(* IEC 61131-3 sources: volt/packages/volt-lsp-iec/test-corpus/pro2193/Device/Plc Logic/Application/09 Misc/Library Manager/L_MC1P_MotionControlBasic (part 3) *)

(* ---- L_MB1P_TPCONVERTTP.pou ---- *)
FUNCTION_BLOCK L_MB1P_TPCONVERTTP
VAR_INPUT
	XENABLE : BOOL;
	XTPRECEIVE : BOOL;
	LRACTTPPOSIN : LREAL;
	LRCYCPOSTPAXIS : LREAL;
	LRCYCPOSTARGETAXIS : LREAL;
	LRCYCLELENGTHTPAXIS : LREAL;
	LRCYCLELENGTHTARGETAXIS : LREAL;
END_VAR
VAR_OUTPUT
	XTPRECEIVED : BOOL;
	LRTPACTPOS : LREAL;
	XERROR : BOOL;
	EERRORID : L_IE1P_Error;
END_VAR
VAR
	LRPOSFIFOX : ARRAY [1..20] OF LREAL := [10(0)];
	LRPOSFIFOREG : ARRAY [1..20] OF LREAL := [10(0)];
	BYCOUNTER : INT := 1;
	LRSTACKDIFFERENCE : LREAL;
	LRTPDELTAINMS : LREAL;
	LRDELTAPCT : LREAL;
	XTPRECEIVEDOLD : BOOL;
	LRTEMP : LREAL;
	IDIRECTION : INT;
	LRACTTPPOSIN_OLD : LREAL;
	XWAIT : BOOL;
	XWAIT_OLD : BOOL;
	LRACTTPPOSIN_INT : LREAL;
	R_TRIG1 : R_TRIG;
END_VAR
END_FUNCTION_BLOCK

METHOD SEARCHINSTACKNEGATIVE
END_METHOD

METHOD SEARCHINSTACKPOSITIVE
END_METHOD

(* ---- L_MB1P_TPTIMESTAMPTOPOS.pou ---- *)
FUNCTION_BLOCK L_MB1P_TPTIMESTAMPTOPOS
VAR_INPUT
	XENABLE : BOOL;
	XTPRECEIVE : BOOL;
	DWTPTIMESTAMP : DWORD;
	LRACTPOSIN : LREAL;
	LRCYCLELENGTH : LREAL;
	DWDELAYACTPOS : DWORD;
END_VAR
VAR_OUTPUT
	XBUSY : BOOL;
	XERROR : BOOL;
	EERRORID : L_IE1P_Error;
	XTPRECEIVED : BOOL;
	LRTPACTPOS : LREAL;
END_VAR
VAR
	XENABLEOLD : BOOL;
	WACTIDX : WORD;
	ALRPOS : ARRAY [0..31] OF LREAL;
	DITIMESTAMPDIFF : DINT;
	DWACTDCTIME : DWORD;
	DWTASKYCLE_NS : DWORD;
	XINIT : BOOL := TRUE;
	LRBASE : LREAL;
	LRDIFF : LREAL;
	LRFACTOR : LREAL;
	LRCAPTURE : LREAL;
	UDIINTERVAL : UDINT;
	LRINTERVAL : LREAL;
	XTPRECEIVEOLD : BOOL;
	C_WMAXELEMENTS : WORD := 31;
END_VAR
END_FUNCTION_BLOCK

METHOD CALCTPPOS : LREAL
END_METHOD

(* ---- L_MC1P_ABORTTRIGGER_INTERNAL.pou ---- *)
FUNCTION_BLOCK L_MC1P_ABORTTRIGGER_INTERNAL EXTENDS L_MC1P_Template_IntFB
VAR_INPUT
	EXECUTE : BOOL;
	PAUSEACTIVETP : BOOL;
END_VAR
VAR_OUTPUT
	DONE : BOOL;
	BUSY : BOOL;
	ERROR : BOOL;
	ERRORID : L_IE1P_Error;
END_VAR
VAR
	PTPREF : POINTER TO L_MC1P_TPData;
	EXECUTEOLD : BOOL := FALSE;
	SNTPNUMBER : SINT;
END_VAR
END_FUNCTION_BLOCK

METHOD MAIN
VAR_IN_OUT
	AXIS : AXIS_REF;
	FBBASE : L_MC1P_Template_ForAxis;
	TRIGGERINPUT : MC_TRIGGER_REF;
END_VAR
END_METHOD

(* ---- L_MC1P_ADDOFFSETCYCLIC.pou ---- *)
FUNCTION_BLOCK L_MC1P_ADDOFFSETCYCLIC
VAR_INPUT
	LRSETPOS : LREAL;
	LRSETOFFSET : LREAL;
	ETRAVERSINGRANGE : L_MC1P_TraversingRange := L_MC1P_TraversingRange.Modulo;
	LRCYCLELENGTH : LREAL;
END_VAR
VAR_OUTPUT
	LRSETPOSOUT : LREAL;
	XERROR : BOOL;
	EERRORID : L_IE1P_Error;
END_VAR
VAR
	LRPOSDIFF : LREAL;
	LRPOS : LREAL;
	LRLENGTH : LREAL;
END_VAR
END_FUNCTION_BLOCK

(* ---- L_MC1P_AVERAGEFILTERSETVALUES.pou ---- *)
FUNCTION_BLOCK L_MC1P_AVERAGEFILTERSETVALUES EXTENDS L_MC1P_SetSetValueManipulator
VAR_INPUT
	WFILTERDEPTH : WORD;
	XMANIPULATETORQUE : BOOL := FALSE;
END_VAR
VAR_OUTPUT
	XINEQOUT : BOOL;
END_VAR
VAR
	WFILTERDEPTHINT : WORD := 20;
	CWFILTERDEPTHMAX : WORD := 1000;
	LRFILTERDEPTH : LREAL;
	LRINVFILTERDEPTH : LREAL;
	WCOUNTER : WORD;
	XERROR_CHECKINPUTDATA : BOOL;
	LRHOMINGOFFSETACT : LREAL;
	LRFILTEREDPOS : LREAL;
	AVERAGEFILTER : L_MC1P_TimeAverage;
	XMANIPULATETORQUEINT : BOOL := FALSE;
END_VAR
END_FUNCTION_BLOCK

METHOD CALCULATE2
VAR_IN_OUT
	AXIS : AXIS_REF;
END_VAR
END_METHOD

METHOD CALLCYCLIC2
VAR_IN_OUT
	AXIS : AXIS_REF;
END_VAR
END_METHOD

METHOD ENABLEINIT2
VAR_IN_OUT
	AXIS : Axis_REf;
END_VAR
END_METHOD

METHOD INITIALIZEFILTER
END_METHOD

METHOD LOADOFFSET2
VAR_INPUT
	OFFSET : LREAL;
END_VAR
VAR_IN_OUT
	AXIS : AXIS_REF;
END_VAR
END_METHOD

METHOD READINPUTS2
VAR_IN_OUT
	AXIS : AXIS_REF;
END_VAR
END_METHOD

(* ---- L_MC1P_AXIS_REF_POOL_2AXES.pou ---- *)
FUNCTION_BLOCK L_MC1P_AXIS_REF_POOL_2AXES
VAR_OUTPUT
	AXESPOOL : L_MC1P_IAXIS_REF_POOL;
END_VAR
VAR_IN_OUT
	AXIS1 : AXIS_REF;
	AXIS2 : AXIS_REF;
END_VAR
VAR
	AAXIS : ARRAY [1..2] OF POINTER TO AXIS_REF;
	WAXISCOUNT : WORD;
	AXISPOOLCOUNT : WORD;
END_VAR
END_FUNCTION_BLOCK

METHOD GETAXISFROMPOOL : POINTER TO AXIS_REF
VAR_INPUT
	WINDEX : WORD;
END_VAR
END_METHOD

(* ---- L_MC1P_AXIS_REF_POOL_3AXES.pou ---- *)
FUNCTION_BLOCK L_MC1P_AXIS_REF_POOL_3AXES
VAR_OUTPUT
	AXESPOOL : L_MC1P_IAXIS_REF_POOL;
END_VAR
VAR_IN_OUT
	AXIS1 : AXIS_REF;
	AXIS2 : AXIS_REF;
	AXIS3 : AXIS_REF;
END_VAR
VAR
	AAXIS : ARRAY [1..3] OF POINTER TO AXIS_REF;
	WAXISCOUNT : WORD;
	AXISPOOLCOUNT : WORD;
END_VAR
END_FUNCTION_BLOCK

METHOD GETAXISFROMPOOL : POINTER TO AXIS_REF
VAR_INPUT
	WINDEX : WORD;
END_VAR
END_METHOD

(* ---- L_MC1P_AXISBASICCONTROL.pou ---- *)
FUNCTION_BLOCK L_MC1P_AXISBASICCONTROL EXTENDS L_MC1P_Template_Licence_150
VAR_INPUT
	XENABLEINTERNALCONTROL : BOOL;
	XREGULATORON : BOOL;
	XRESETERROR : BOOL;
	XENABLEPOSITIVE : BOOL := TRUE;
	XENABLENEGATIVE : BOOL := TRUE;
	XDISABLESWLIMIT : BOOL := FALSE;
	LROVERRIDE : LREAL := 1.0;
	LROVERRIDEACC : LREAL := 1.0;
	LROVERRIDEJERK : LREAL := 1.0;
	XSTOP : BOOL;
	LRSTOPDEC : LREAL := 360000;
	LRSTOPJERK : LREAL := 0;
	XJOGGINGPOS : BOOL;
	XJOGGINGNEG : BOOL;
	LRJOGGINGSETVEL : LREAL := 3600;
	LRJOGGINGSETACC : LREAL := 36000;
	LRJOGGINGSETDEC : LREAL := 36000;
	LRJOGGINGSETJERK : LREAL := 0;
	XCONTINUOUSUPDATE : BOOL;
	XMOVEVELEXECUTE : BOOL;
	XMOVEABSEXECUTE : BOOL;
	XMOVERELEXECUTE : BOOL;
	XHALT : BOOL;
	LRSETPOS_DIST : LREAL;
	LRSETVEL : LREAL := 3600;
	LRSETACC : LREAL := 36000;
	LRSETDEC : LREAL := 36000;
	LRSETJERK : LREAL := 0;
	ESETDIRECTION : MC_DIRECTION := MC_DIRECTION.mcPositiveDirection;
	XHOMEEXECUTE : BOOL;
	LRHOMEPOSITION : LREAL;
	XUSEHOMEEXTPARAMETER : BOOL;
	SCHOMEEXTPARAMETER : L_MC1P_HomeParameter;
	SCHOMEEXTTP : MC_TRIGGER_REF;
	XHOMEABSSWITCH : BOOL;
END_VAR
VAR_OUTPUT
	XINTERNALCONTROLACTIVE : BOOL;
	XERROR : BOOL;
	EERRORID : L_IE1P_Error;
	XFUNBUSY : BOOL;
	XFUNDONE : BOOL;
	XFUNCOMMANDABORTED : BOOL;
	EFUNSTATEACT : L_MC1P_ABC_State;
	ECONTROLMODE : L_MC1P_ControlMode;
	XISHOMED : BOOL;
	XHWLIMITSWITCHNEG : BOOL;
	XHWLIMITSWITCHPOS : BOOL;
	XSWLIMITENABLED : BOOL;
	XSWLIMITSWITCHNEG : BOOL;
	XSWLIMITSWITCHPOS : BOOL;
	EAXISTYPE : L_MC1P_DriveType;
	EAXISSTATE : L_MC1P_AXIS_STATE := L_MC1P_AXIS_STATE.Disabled;
	XAXISREADY : BOOL;
	XAXISENABLED : BOOL;
	XAXISWARNING : BOOL;
	XAXISERROR : BOOL;
	EAXISERRORID : L_IE1P_Error;
	XDRIVEWARNING : BOOL;
	XDRIVEERROR : BOOL;
	DWDRIVEERRORID : DWORD;
	LRACTPOS : LREAL;
	LRACTVEL : LREAL;
	LRSETPOSOUT : LREAL;
	LRSETVELOUT : LREAL;
	LRACTFOLLOWINGERROR : LREAL;
	XCONSTANTVELOCITY : BOOL;
	XACCELERATING : BOOL;
	XDECELERATING : BOOL;
	XDIRECTIONPOSITIVE : BOOL;
	XDIRECTIONNEGATIVE : BOOL;
	XINPOSITION : BOOL;
	XAXISAVAILABLE : BOOL;
	XSTANDSTILLSETVELOCITY : BOOL;
	XSTANDSTILLACTVELOCITY : BOOL;
	XAXISREADYTOSWITCHON : BOOL;
	XAXISREADYFORMOTION : BOOL;
END_VAR
VAR
	XREGULATORON_INT : BOOL;
	XRESETERROR_INT : BOOL;
	XENABLEPOSITIVE_INT : BOOL;
	XENABLENEGATIVE_INT : BOOL;
	XDISABLESWLIMIT_INT : BOOL;
	LROVERRIDE_INT : LREAL := 1.0;
	LROVERRIDEACC_INT : LREAL := 1.0;
	LROVERRIDEJERK_INT : LREAL := 1.0;
	XSTOP_INT : BOOL;
	LRSTOPDEC_INT : LREAL;
	LRSTOPJERK_INT : LREAL;
	XHALT_INT : BOOL;
	XJOGGINGPOS_INT : BOOL;
	XJOGGINGNEG_INT : BOOL;
	LRJOGGINGSETVEL_INT : LREAL;
	LRJOGGINGSETACC_INT : LREAL;
	LRJOGGINGSETDEC_INT : LREAL;
	LRJOGGINGSETJERK_INT : LREAL := 0;
	LRJOGGINGSETJERKDEC_INT : LREAL := 0;
	LRJOGGINGSETJERKDECAPP : LREAL := 0;
	XMOVEVELEXECUTE_INT : BOOL;
	XMOVEABSEXECUTE_INT : BOOL;
	XMOVERELEXECUTE_INT : BOOL;
	XCONTINUOUSUPDATE_INT : BOOL;
	LRSETPOS_DIST_INT : LREAL;
	LRSETVEL_INT : LREAL;
	LRSETACC_INT : LREAL;
	LRSETDEC_INT : LREAL;
	LRSETJERK_INT : LREAL;
	LRSETJERKDEC_INT : LREAL := 0;
	LRSETJERKDECAPP : LREAL := 0;
	ESETDIRECTION_INT : MC_DIRECTION;
	XHOMEEXECUTE_INT : BOOL;
	LRHOMEPOSITION_INT : LREAL;
	XHOMEEXTERNALVALUES_INT : BOOL;
	SCHOMEEXTPARAMETER_INT : L_MC1P_HomeParameter;
	XDISABLEMOVEFUNEXEC : BOOL;
	XINTERNALCONTROLVISU : BOOL;
	XDISABLEMOVEFUN : BOOL;
	XDISABLEHOMEFUN : BOOL;
	XDISABLEPOWERFUN : BOOL;
	XDISABLEPOWERCALL : BOOL;
	XVISUMOVEFUN : BOOL;
	XVISUHOMEFUN : BOOL;
	XVISUPOWFUN : BOOL;
	ABC : REFERENCE TO L_MC1P_AxisBasicControl_Internal;
	DATA : L_MC1P_AxisBasicControlInstanceData;
	FBBASEOLD : POINTER TO L_MC1P_Template_ForAxis;
	_USEQSP : BOOL := FALSE;
	DISABLEHOMEFUN : BOOL;
	DISABLEMOVEFUN : BOOL;
	DISABLEMOVEFUNEXEC : BOOL;
	DISABLEPOWERCALL : BOOL;
	DISABLEPOWERFUN : BOOL;
	LRJOGGINGSETJERKDEC : LREAL;
	LRSETJERKDEC : LREAL;
	USEQSP : BOOL;
END_VAR
END_FUNCTION_BLOCK

(* ---- L_MC1P_AXISBASICCONTROL_INTERNAL.pou ---- *)
FUNCTION_BLOCK L_MC1P_AXISBASICCONTROL_INTERNAL EXTENDS L_MC1P_Template_IntFB
VAR_INPUT
	XDISABLEPOWERCALL : BOOL;
	XREGULATORON : BOOL;
	XRESETERROR : BOOL;
	XENABLEPOSITIVE : BOOL := TRUE;
	XENABLENEGATIVE : BOOL := TRUE;
	XDISABLESWLIMIT : BOOL;
	LROVERRIDE : LREAL := 1.0;
	LROVERRIDEACC : LREAL := 1.0;
	LROVERRIDEJERK : LREAL := 1.0;
	XSTOP : BOOL;
	LRSTOPDEC : LREAL;
	LRSTOPJERK : LREAL;
	XJOGGINGPOS : BOOL;
	XJOGGINGNEG : BOOL;
	LRJOGGINGSETVEL : LREAL := 3600;
	LRJOGGINGSETACC : LREAL := 36000;
	LRJOGGINGSETDEC : LREAL := 36000;
	LRJOGGINGSETJERK : LREAL := 0;
	LRJOGGINGSETJERKDEC : LREAL := 0;
	XCONTINUOUSUPDATE : BOOL;
	XFINISHPOSITIONING : BOOL;
	XQSPAPPLICATION : BOOL;
	XHALT : BOOL;
	XABORT : BOOL;
	XMOVEVELEXECUTE : BOOL;
	XMOVEABSEXECUTE : BOOL;
	XMOVERELEXECUTE : BOOL;
	LRSETPOS_DIST : LREAL;
	LRSETVEL : LREAL := 3600;
	LRSETACC : LREAL := 36000;
	LRSETDEC : LREAL := 36000;
	LRSETJERK : LREAL := 0;
	LRSETJERKDEC : LREAL := 0;
	ESETDIRECTION : MC_DIRECTION := MC_DIRECTION.mcPositiveDirection;
	XHOMEEXECUTE : BOOL;
	LRHOMEPOSITION : LREAL;
	XUSEHOMEEXTPARAMETER : BOOL;
	SCHOMEEXTPARAMETER : L_MC1P_HomeParameter;
	SCHOMEEXTTP : MC_TRIGGER_REF;
	XHOMEABSSWITCH : BOOL;
	XRESETHOMEPOSITION : BOOL;
	WCALLEDINCYCLE : WORD;
	XQSPDRIVEDONE : BOOL;
	XMOVEVELENABLEOFFSETVEL : BOOL;
	LRMOVEVELOFFSETVEL : LREAL;
	XUSEABORTBEHAVIOURFORTM : BOOL;
	LRABORTDEC : LREAL;
	LRABORTJERK : LREAL;
END_VAR
VAR_OUTPUT
	ECONTROLMODE : L_MC1P_ControlMode;
	XISHOMED : BOOL;
	XHWLIMITSWITCHNEG : BOOL;
	XHWLIMITSWITCHPOS : BOOL;
	XSWLIMITENABLED : BOOL;
	XSWLIMITSWITCHNEG : BOOL;
	XSWLIMITSWITCHPOS : BOOL;
	EAXISTYPE : L_MC1P_DriveType;
	EAXISSTATE : L_MC1P_AXIS_STATE := L_MC1P_AXIS_STATE.Disabled;
	XAXISREADY : BOOL;
	XAXISENABLED : BOOL;
	XAXISWARNING : BOOL;
	XAXISERROR : BOOL;
	EAXISERRORID : L_IE1P_Error;
	XDRIVEWARNING : BOOL;
	XDRIVEERROR : BOOL;
	DWDRIVEERRORID : DWORD;
	LRACTPOS : LREAL;
	LRACTVEL : LREAL;
	LRSETPOSOUT : LREAL;
	LRSETVELOUT : LREAL;
	LRACTFOLLOWINGERROR : LREAL;
	XCONSTANTVELOCITY : BOOL;
	XACCELERATING : BOOL;
	XDECELERATING : BOOL;
	XDIRECTIONPOSITIVE : BOOL;
	XDIRECTIONNEGATIVE : BOOL;
	XINPOSITION : BOOL;
	XAXISAVAILABLE : BOOL;
	XSTANDSTILLSETVELOCITY : BOOL;
	XSTANDSTILLACTVELOCITY : BOOL;
	XAXISREADYTOSWITCHON : BOOL;
	XAXISREADYFORMOTION : BOOL;
END_VAR
VAR
	ABCFUNID : WORD;
	FBSTOP : L_MC1P_Stop_Internal;
	FBHALT : L_MC1P_Halt_Internal;
	FBABORT : L_MC1P_Halt_Internal;
	FBHOME : L_MC1P_Home_Internal;
	FBJOG : L_MC1P_ManualJog_Internal;
	FBMOVEABS : L_MC1P_MoveAbsolute_Inernal;
	FBMOVEVEL : L_MC1P_MoveVelocity_Internal;
	FBMOVEREL : L_MC1P_MoveRelative_Internal;
	FBFINISHPOSITIONING : L_MC1P_FinishPositioning_internal;
	PBDUMMY : POINTER TO BOOL;
	XCONTROLLEDBYAXIS : BOOL;
	XCALLEDBYAXIS : BOOL;
	XUPDATESTATE : BOOL;
	XUPDATECONTROL : BOOL;
	XDISABLEMOVEFUNEXEC : BOOL;
	XDISABLEINTERNALCALLOFMOVEFUNCTIONS : BOOL;
	ETMPHOMEMODE : L_MC1P_HomeMode;
	LRTMPOFFSETPOSITION : LREAL;
	AXISCONTROL : BOOL;
	CALLEDBYAXIS : BOOL;
	DISABLEMOVEFUNEXEC : BOOL;
END_VAR
END_FUNCTION_BLOCK

METHOD BASEITFCHANGED
VAR_INPUT
	FBBASEOLD : POINTER TO POINTER TO L_MC1P_Template_ForAxis;
END_VAR
VAR_IN_OUT
	AXIS : AXIS_REF;
	FBBASE : L_MC1P_Template_ForAxis;
	DATA : L_MC1P_AxisBasicControlInstanceData;
END_VAR
END_METHOD

METHOD CALLMOVEFB : BOOL
VAR_IN_OUT
	AXIS : AXIS_REF;
	DATA : L_MC1P_AxisBasicControlInstanceData;
END_VAR
END_METHOD

METHOD EXITSTATE
VAR_IN_OUT
	AXIS : AXIS_REF;
	DATA : L_MC1P_AxisBasicControlInstanceData;
END_VAR
END_METHOD

METHOD MAIN
VAR_IN_OUT
	AXIS : AXIS_REF;
	FBBASE : L_MC1P_Template_ForAxis;
	DATA : L_MC1P_AxisBasicControlInstanceData;
END_VAR
END_METHOD

METHOD RESET
VAR_IN_OUT
	DATA : L_MC1P_AxisBasicControlInstanceData;
END_VAR
END_METHOD

METHOD RESETACTIVEINSTANCE : WORD
END_METHOD

METHOD SETACTIVEINSTANCE : WORD
END_METHOD

METHOD STATEMACHINE
VAR_IN_OUT
	AXIS : AXIS_REF;
	DATA : L_MC1P_AxisBasicControlInstanceData;
END_VAR
END_METHOD

(* ---- L_MC1P_AXISBASICCONTROLV2.pou ---- *)
FUNCTION_BLOCK L_MC1P_AXISBASICCONTROLV2 EXTENDS L_MC1P_Template_Licence_150
VAR_INPUT
	XENABLEINTERNALCONTROL : BOOL;
	XENABLEOPERATION : BOOL;
	XRESETERROR : BOOL;
	XENABLEPOSITIVE : BOOL := TRUE;
	XENABLENEGATIVE : BOOL := TRUE;
	XDISABLESWLIMIT : BOOL := FALSE;
	LROVERRIDE : LREAL := 1.0;
	LROVERRIDEACC : LREAL := 1.0;
	LROVERRIDEJERK : LREAL := 1.0;
	XQSPAPPLICATION : BOOL;
	XHALT : BOOL;
	XABORT : BOOL;
	XJOGPOS : BOOL;
	XJOGNEG : BOOL;
	XCONTINUOUSUPDATE : BOOL;
	XFINISHPOSITIONING : BOOL;
	XMOVEVELEXECUTE : BOOL;
	XMOVEABSEXECUTE : BOOL;
	XMOVERELEXECUTE : BOOL;
	LRPOS_DIST : LREAL := 0;
	LRVEL : LREAL := 3600;
	LRACC : LREAL := 36000;
	LRDEC : LREAL := 36000;
	LRJERK : LREAL := 0;
	EDIRECTION : MC_DIRECTION := MC_DIRECTION.mcPositiveDirection;
	XHOMEEXECUTE : BOOL;
	SCHOMEEXTTP : MC_TRIGGER_REF;
	XHOMEABSSWITCH : BOOL;
	XRESETHOMEPOSITION : BOOL;
END_VAR
VAR_OUTPUT
	XINTERNALCONTROLACTIVE : BOOL;
	XERROR : BOOL;
	EERRORID : L_IE1P_Error;
	XFUNBUSY : BOOL;
	XFUNDONE : BOOL;
	XFUNCOMMANDABORTED : BOOL;
	EFUNSTATEACT : L_MC1P_ABC_State := L_MC1P_ABC_State.Standby;
	ECONTROLMODE : L_MC1P_ControlMode := L_MC1P_ControlMode.PosCtrlDrive;
	XISHOMED : BOOL;
	XHWLIMITSWITCHNEG : BOOL;
	XHWLIMITSWITCHPOS : BOOL;
	XSWLIMITENABLED : BOOL;
	XSWLIMITSWITCHNEG : BOOL;
	XSWLIMITSWITCHPOS : BOOL;
	EAXISTYPE : L_MC1P_DriveType := L_MC1P_DriveType.Virtual;
	EAXISSTATE : L_MC1P_AXIS_STATE := L_MC1P_AXIS_STATE.Disabled;
	XSTOACTIVE : BOOL;
	XREADYFOROPERATION : BOOL;
	XOPERATIONENABLED : BOOL;
	XREADYFORMOTION : BOOL;
	XAXISWARNING : BOOL;
	XAXISERROR : BOOL;
	EAXISERRORID : L_IE1P_Error;
	XDRIVEWARNING : BOOL;
	XDRIVEERROR : BOOL;
	DWDRIVEERRORID : DWORD;
	LRACTPOS : LREAL;
	LRACTVEL : LREAL;
	LRSETPOSOUT : LREAL;
	LRSETVELOUT : LREAL;
	LRACTFOLLOWINGERROR : LREAL;
	XINPOSITION : BOOL;
	XSTANDSTILLSETVELOCITY : BOOL;
	XSTANDSTILLACTVELOCITY : BOOL;
	XCONSTANTVELOCITY : BOOL;
	XACCELERATING : BOOL;
	XDECELERATING : BOOL;
	XDIRECTIONPOSITIVE : BOOL;
	XDIRECTIONNEGATIVE : BOOL;
	XAXISAVAILABLE : BOOL;
END_VAR
VAR
	_ITFOWNER : L_UBUP.L_UBUP_IFBPool;
	_XWHANDLE : __XWORD;
	_XOCCUPIED : BOOL;
	XENABLEOPERATION_INT : BOOL;
	XRESETERROR_INT : BOOL;
	XENABLEPOSITIVE_INT : BOOL;
	XENABLENEGATIVE_INT : BOOL;
	XDISABLESWLIMIT_INT : BOOL;
	LROVERRIDE_INT : LREAL;
	LROVERRIDEACC_INT : LREAL;
	LROVERRIDEJERK_INT : LREAL;
	XQSPAPPLICATION_INT : BOOL;
	XHALT_INT : BOOL;
	XABORT_INT : BOOL;
	XJOGPOS_INT : BOOL;
	XJOGNEG_INT : BOOL;
	XCONTINUOUSUPDATE_INT : BOOL;
	XFINISHPOSITIONING_INT : BOOL;
	XMOVEVELEXECUTE_INT : BOOL;
	XMOVEABSEXECUTE_INT : BOOL;
	XMOVERELEXECUTE_INT : BOOL;
	LRPOS_DIST_INT : LREAL;
	LRVEL_INT : LREAL;
	LRACC_INT : LREAL;
	LRDEC_INT : LREAL;
	LRJERK_INT : LREAL;
	EDIRECTION_INT : MC_DIRECTION;
	XHOMEEXECUTE_INT : BOOL;
	XRESETHOMEPOSITION_INT : BOOL;
	LRSETJERKDEC_INT : LREAL;
	LRJOGGINGSETJERKDEC_INT : LREAL;
	LRSETJERKDECAPP : LREAL;
	LRJOGGINGSETJERKDECAPP : LREAL;
	XDISABLEMOVEFUNEXEC : BOOL;
	XDISABLEPOWERCALL : BOOL;
	XINTERNALCONTROLVISU : BOOL;
	XDISABLEMOVEFUN : BOOL;
	XDISABLEHOMEFUN : BOOL;
	XDISABLEPOWERFUN : BOOL;
	XVISUMOVEFUN : BOOL;
	XVISUHOMEFUN : BOOL;
	XVISUPOWFUN : BOOL;
	LRMOVEVELOFFSETVELAPP : LREAL;
	XMOVEVELENABLEOFFSETVELAPP : BOOL;
	LRABORTDECAPP : LREAL;
	LRABORTJERKAPP : LREAL;
	XUSEABORTBEHAVIOURFORTM : BOOL;
	ABC : REFERENCE TO L_MC1P_AxisBasicControl_Internal;
	DATA : L_MC1P_AxisBasicControlInstanceData;
	FBBASEOLD : POINTER TO L_MC1P_Template_ForAxis;
	_DWOBJID : DWORD;
	CLASSID : DINT;
	DISABLEHOMEFUN : BOOL;
	DISABLEMOVEFUN : BOOL;
	DISABLEMOVEFUNEXEC : BOOL;
	DISABLEPOWERCALL : BOOL;
	DISABLEPOWERFUN : BOOL;
	INSTANCEPTR : POINTER TO BYTE;
	LRABORTDEC : LREAL;
	LRABORTJERK : LREAL;
	LRJOGGINGSETJERKDEC : LREAL;
	LRMOVEVELOFFSETVEL : LREAL;
	LRSETJERKDEC : LREAL;
	OBJECTID : DWORD;
	OCCUPIED : BOOL;
	REMAININGTIMEOFPROFILE : LREAL;
	REMAININGTIMEOFPROFILEAVAILABLE : BOOL;
	XMOVEVELENABLEOFFSETVEL : BOOL;
	XSPECIALABORTBEHAVIOR : BOOL;
END_VAR
END_FUNCTION_BLOCK

METHOD RESETABORT
END_METHOD

METHOD RESETFINISHPOSITIONING
END_METHOD

METHOD RESETHALT
END_METHOD

METHOD RESETHOMEEXECUTE
END_METHOD

METHOD RESETMOVEABSEXECUTE
END_METHOD

METHOD RESETMOVERELEXECUTE
END_METHOD

METHOD RESETMOVEVELEXECUTE
END_METHOD

METHOD FREE : BOOL
END_METHOD

METHOD OCCUPY : BOOL
VAR_INPUT
	ITFOWNER : L_UBUP.L_UBUP_IFBPool;
	XWHANDLE : __XWORD;
END_VAR
END_METHOD

METHOD REQUESTINTERFACE : BOOL
VAR_INPUT
	ID : DINT;
	PITFUNKNOWN : POINTER TO L_UBUP_IUnknown;
END_VAR
END_METHOD

METHOD FB_INIT : BOOL
VAR_INPUT
	BINITRETAINS : BOOL;
	BINCOPYCODE : BOOL;
END_VAR
END_METHOD

(* ---- L_MC1P_AXISCOMMAND.pou ---- *)
FUNCTION_BLOCK L_MC1P_AXISCOMMAND
VAR_INPUT
	COMMANDIN : USINT;
END_VAR
VAR_OUTPUT
	XCOMMANDBUSY : BOOL;
END_VAR
VAR
	XABORT : BOOL;
	COMMAND : REFERENCE TO USINT;
	COMMANDOLD : USINT;
	FB_BASE : L_MC1P_Template_ForAxis;
	C_CMDREADY : USINT := 0;
	C_CMDSTART : USINT := 1;
	C_CMDINPROGRESS : USINT := 2;
	C_CMDCANCELLED : USINT := 3;
	C_CMDNOACCESS : USINT := 4;
	C_CMDNOACCESSDISABLED : USINT := 5;
	C_CMDABORT : USINT := 16;
	C_CMDWORKING20 : USINT := 20;
	C_CMDWORKING40 : USINT := 40;
	C_CMDWORKING60 : USINT := 60;
	C_CMDWORKING80 : USINT := 80;
	C_CMDWRONGBRAKEMODE : USINT := 101;
	C_CMDSTOACTIVE : USINT := 102;
	C_CMDINVALIDPARAMETERSETTINGS : USINT := 103;
	C_CMDSTARTOUTSIDEPOSLIMITS : USINT := 104;
	C_CMDPOSRANGENOTSUFFICIENT : USINT := 105;
	C_CMDHOMEPOSREQUIRED : USINT := 106;
	C_CMDINVALIDPOSITIONLIMITS : USINT := 107;
	C_CMDVIRTUALMODENOTSUPPORTED : USINT := 120;
	BUSY : BOOL;
END_VAR
END_FUNCTION_BLOCK

METHOD ABORTING
END_METHOD

METHOD CALCSTATUS
VAR_IN_OUT
	AXIS : _AXIS_REF_REAL;
END_VAR
END_METHOD

METHOD EXECUTE
END_METHOD

METHOD MAIN
END_METHOD

METHOD READINPUTS
END_METHOD

METHOD RESETCOMMANDERRORSTATE : BOOL
VAR_IN_OUT
	AXIS : _AXIS_REF_REAL;
END_VAR
END_METHOD

METHOD RESETSTATUSPARAMETER
END_METHOD

METHOD SETINCTANCEINFO
VAR_INPUT
	PSINSTANCENAME : POINTER TO STRING;
	ERRORITFID : DWORD;
END_VAR
END_METHOD

METHOD UPDATEAXISPOINTER
VAR_INPUT
	PAXIS : POINTER TO AXIS_REF;
END_VAR
END_METHOD

METHOD UPDATECOMMANDINTERFACE
VAR_IN_OUT
	CMD : USINT;
END_VAR
END_METHOD

METHOD FB_INIT : BOOL
VAR_INPUT
	BINITRETAINS : BOOL;
	BINCOPYCODE : BOOL;
END_VAR
END_METHOD

(* ---- L_MC1P_AXISCOMMAND_BRAKEGRINDIN.pou ---- *)
FUNCTION_BLOCK L_MC1P_AXISCOMMAND_BRAKEGRINDIN EXTENDS L_MC1P_AxisCommand
VAR_INPUT
	PAXIS : POINTER TO _AXIS_REF_REAL;
	EMODE : L_MC1P_GrindInMode := L_MC1P_GrindInMode.CwCcw;
	LRMOTORSPEED : LREAL := 60.0;
	LRRAMPTIME : LREAL := 1.0;
	LRONTIME : LREAL := 0.5;
	LROFFTIME : LREAL := 0.5;
	WCYCLES : WORD := 4;
	USICONTROL : USINT;
END_VAR
VAR
	FB_BRAKEGRINDIN : L_MC1P_BrakeGrindIn_internal;
	STATUS_100 : LREAL;
	LRSTATUS : LREAL;
	C_WSTATESUCCESSFUL : WORD := 10;
	C_WSTATEABORTEDERROR : WORD := 8;
	C_WSTATEABORTEDUSER : WORD := 9;
END_VAR
END_FUNCTION_BLOCK

METHOD ABORTING
END_METHOD

METHOD EXECUTE
END_METHOD

METHOD READINPUTS
END_METHOD

METHOD RESETSTATUSPARAMETER
END_METHOD

METHOD UPDATEAXISPOINTER
VAR_INPUT
	PAXIS : POINTER TO AXIS_REF;
END_VAR
END_METHOD

(* ---- L_MC1P_AXISCOMMAND_BRAKETEST.pou ---- *)
FUNCTION_BLOCK L_MC1P_AXISCOMMAND_BRAKETEST EXTENDS L_MC1P_AxisCommand
VAR_INPUT
	PAXIS : POINTER TO _AXIS_REF_REAL;
END_VAR
VAR
	FB_BRAKETEST : L_MC1P_BrakeTest_internal;
	ACTPOSTHRESHOLD : INT;
	STATUS_100 : LREAL;
	LRSTATUS : LREAL;
	LRTIME : LREAL;
	C_WSTATESUCCESSFUL : WORD := 10;
	C_WSTATEFAILED : WORD := 11;
	C_WSTATEABORTEDERROR : WORD := 8;
	C_WSTATEABORTEDUSER : WORD := 9;
END_VAR
END_FUNCTION_BLOCK

METHOD ABORTING
END_METHOD

METHOD EXECUTE
END_METHOD

METHOD READINPUTS
END_METHOD

METHOD RESETSTATUSPARAMETER
END_METHOD

METHOD UPDATEAXISPOINTER
VAR_INPUT
	PAXIS : POINTER TO AXIS_REF;
END_VAR
END_METHOD

(* ---- L_MC1P_AXISCONNECTIONVIEWER.pou ---- *)
FUNCTION_BLOCK L_MC1P_AXISCONNECTIONVIEWER EXTENDS L_IF1P_FunctionConnectionViewer
END_FUNCTION_BLOCK

METHOD BUILDUPCONNECTIONTABLE : BOOL
END_METHOD

METHOD FINDCONNECTIONSOURCE : POINTER TO BYTE
VAR_INPUT
	PSLAVECONNECTOR : POINTER TO IoConfigConnector;
	UITYPE : UINT;
	UISUBDEVICE : UINT;
END_VAR
END_METHOD

METHOD FINDFUNCTION : L_IF1P_IFunctionConnection
VAR_INPUT
	PFUNCTIONCONNECTOR : POINTER TO IoConfigConnector;
END_VAR
VAR_OUTPUT
	UITYPE : UINT;
END_VAR
END_METHOD

METHOD GETCONNECTEDSLAVE : BOOL
END_METHOD

METHOD INITIALIZE : UDINT
VAR_INPUT
	WMODULETYPE : UINT;
	DWINSTANCE : UDINT;
	PCONNECTOR : POINTER TO IoConfigConnector;
END_VAR
END_METHOD

METHOD IODRVREADPARAMETER : UDINT
VAR_INPUT
	PCONNECTOR : POINTER TO IoConfigConnector;
	PPARAMETER : POINTER TO IoConfigParameter;
	PDATA : POINTER TO BYTE;
	DWBITSIZE : DWORD;
	DWBITOFFSET : DWORD;
END_VAR
END_METHOD

METHOD IODRVUPDATECONFIGURATION : UDINT
VAR_INPUT
	PCONNECTORLIST : POINTER TO IoConfigConnector;
	NCOUNT : DINT;
END_VAR
END_METHOD

METHOD IODRVUPDATEMAPPING : UDINT
VAR_INPUT
	PTASKMAPLIST : POINTER TO IoConfigTaskMap;
	NCOUNT : DINT;
END_VAR
END_METHOD

METHOD IODRVWRITEPARAMETER : UDINT
VAR_INPUT
	PCONNECTOR : POINTER TO IoConfigConnector;
	PPARAMETER : POINTER TO IoConfigParameter;
	PDATA : POINTER TO BYTE;
	DWBITSIZE : DWORD;
	DWBITOFFSET : DWORD;
END_VAR
END_METHOD

METHOD QUERYINTERFACE : POINTER TO POINTER TO BYTE
VAR_INPUT
	IID : DWORD;
	PRESULT : POINTER TO UDINT;
END_VAR
END_METHOD

METHOD STATUSCHANGED : BOOL
END_METHOD

METHOD FB_EXIT : BOOL
VAR_INPUT
	BINCOPYCODE : BOOL;
END_VAR
END_METHOD

METHOD FB_INIT : BOOL
VAR_INPUT
	BINITRETAINS : BOOL;
	BINCOPYCODE : BOOL;
END_VAR
END_METHOD

METHOD EVENTCALLBACK : UDINT
VAR_INPUT
	PEVENTPARAM : POINTER TO EventParam;
END_VAR
END_METHOD

METHOD REGISTEREVENT
END_METHOD

METHOD UNREGISTEREVENT
END_METHOD

(* ---- L_MC1P_AXISEXTENSION_9400HL.pou ---- *)
FUNCTION_BLOCK L_MC1P_AXISEXTENSION_9400HL EXTENDS L_MC1P_AxisExtensionEmpty
VAR
	ECATCOMM : L_MC1P_CommECAT;
	CONFIGDRIVE : L_MC1P_Config_94HL_ETC;
	DRIVESCALING : L_MC1P_DriveScaling_94HL;
	DRIVESPECIFIC : L_MC1P_DriveSpecific_9400HL;
	FBEXTENDEDMAPPINGACCESS : L_MC1P_ExtendedMappingAccess;
	ITFCOMM : L_MC1P_ICommunication;
	ITFCONFIGDRIVE : L_MC1P_IConfigureDrive;
	ITFDRIVESCALING : L_MC1P_IDriveScaling;
	ITFDRIVESPECIFIC : L_MC1P_IDriveSpecificImplBase;
	ITFEXTENDEDMAPPINGACCESS : L_MC1P_IExtendedMappingAccess;
END_VAR
END_FUNCTION_BLOCK

(* ---- L_MC1P_AXISEXTENSION_9400HL_CAN.pou ---- *)
FUNCTION_BLOCK L_MC1P_AXISEXTENSION_9400HL_CAN EXTENDS L_MC1P_AxisExtensionEmpty
VAR
	CANCOMM : L_MC1P_CommCAN;
	CONFIGDRIVE : L_MC1P_Config_94HL_ETC;
	DRIVESCALING : L_MC1P_DriveScaling_94HL;
	DRIVESPECIFIC : L_MC1P_DriveSpecific_9400HL;
	FBEXTENDEDMAPPINGACCESS : L_MC1P_ExtendedMappingAccess;
	ITFCOMM : L_MC1P_ICommunication;
	ITFCONFIGDRIVE : L_MC1P_IConfigureDrive;
	ITFDRIVESCALING : L_MC1P_IDriveScaling;
	ITFDRIVESPECIFIC : L_MC1P_IDriveSpecificImplBase;
	ITFEXTENDEDMAPPINGACCESS : L_MC1P_IExtendedMappingAccess;
END_VAR
END_FUNCTION_BLOCK

(* ---- L_MC1P_AXISEXTENSION_ENCBPB.pou ---- *)
FUNCTION_BLOCK L_MC1P_AXISEXTENSION_ENCBPB EXTENDS L_MC1P_AxisExtensionEmpty
VAR
	DRIVESPECIFIC : L_MC1P_DriveSpecific_Enc_Bpb;
	DRIVESCALING : L_MC1P_DriveScaling;
	ITFDRIVESCALING : L_MC1P_IDriveScaling;
	ITFDRIVESPECIFIC : L_MC1P_IDriveSpecificImplBase;
END_VAR
END_FUNCTION_BLOCK

(* ---- L_MC1P_AXISEXTENSION_ENCFREE.pou ---- *)
FUNCTION_BLOCK L_MC1P_AXISEXTENSION_ENCFREE EXTENDS L_MC1P_AxisExtensionEmpty
VAR
	DRIVESPECIFIC : L_MC1P_DriveSpecific_Enc_Free;
	DRIVESCALING : L_MC1P_DriveScaling;
	ITFDRIVESCALING : L_MC1P_IDriveScaling;
	ITFDRIVESPECIFIC : L_MC1P_IDriveSpecificImplBase;
END_VAR
END_FUNCTION_BLOCK

(* ---- L_MC1P_AXISEXTENSION_ENCI500.pou ---- *)
FUNCTION_BLOCK L_MC1P_AXISEXTENSION_ENCI500 EXTENDS L_MC1P_AxisExtensionEmpty
VAR
	I500COMM : L_MC1P_CommECAT;
	DRIVESPECIFIC : L_MC1P_DriveSpecific_Enc_i500;
	DRIVESCALING : L_MC1P_DriveScaling;
	ITFCOMM : L_MC1P_ICommunication;
	ITFDRIVESCALING : L_MC1P_IDriveScaling;
	ITFDRIVESPECIFIC : L_MC1P_IDriveSpecificImplBase;
END_VAR
END_FUNCTION_BLOCK

(* ---- L_MC1P_AXISEXTENSION_ENCI900_ECAT.pou ---- *)
FUNCTION_BLOCK L_MC1P_AXISEXTENSION_ENCI900_ECAT EXTENDS L_MC1P_AxisExtensionEmpty
VAR
	CONFIGAXIS : L_MC1P_Config_i900_Enc_Drive;
	I900COMM : L_MC1P_CommECAT;
	FBEXTENDEDMAPPINGACCESS : L_MC1P_ExtendedMappingAccess;
	DRIVESPECIFIC : L_MC1P_DriveSpecific_Enc_i950 := STRUCT(xCheckCommunicationState := TRUE);
	DRIVESCALING : L_MC1P_DriveScaling_Enci900;
	ITFCOMM : L_MC1P_ICommunication;
	ITFCONFIGDRIVE : L_MC1P_IConfigureDrive;
	ITFDRIVESCALING : L_MC1P_IDriveScaling;
	ITFDRIVESPECIFIC : L_MC1P_IDriveSpecificImplBase;
	ITFEXTENDEDMAPPINGACCESS : L_MC1P_IExtendedMappingAccess;
END_VAR
END_FUNCTION_BLOCK

(* ---- L_MC1P_AXISEXTENSION_ENCI900_TARGET.pou ---- *)
FUNCTION_BLOCK L_MC1P_AXISEXTENSION_ENCI900_TARGET EXTENDS L_MC1P_AxisExtensionEmpty
VAR_INPUT
	COMM : L_MC1P_Commi900;
	CONFIG : L_MC1P_Config_i900_Enc_Drive;
END_VAR
VAR
	DRIVESPECIFIC : L_MC1P_DriveSpecific_Enc_i950;
	DRIVESCALING : L_MC1P_DriveScaling_Enci900;
	ITFCOMM : L_MC1P_ICommunication;
	ITFCONFIGDRIVE : L_MC1P_IConfigureDrive;
	ITFDRIVESCALING : L_MC1P_IDriveScaling;
	ITFDRIVESPECIFIC : L_MC1P_IDriveSpecificImplBase;
END_VAR
END_FUNCTION_BLOCK

(* ---- L_MC1P_AXISEXTENSION_ENCIOETC.pou ---- *)
FUNCTION_BLOCK L_MC1P_AXISEXTENSION_ENCIOETC EXTENDS L_MC1P_AxisExtensionEmpty
VAR
	DRIVESPECIFIC : L_MC1P_DriveSpecific_Enc_IOETC;
	DRIVESCALING : L_MC1P_DriveScaling;
	ITFDRIVESCALING : L_MC1P_IDriveScaling;
	ITFDRIVESPECIFIC : L_MC1P_IDriveSpecificImplBase;
END_VAR
END_FUNCTION_BLOCK

(* ---- L_MC1P_AXISEXTENSION_GENERICDRIVE.pou ---- *)
FUNCTION_BLOCK L_MC1P_AXISEXTENSION_GENERICDRIVE EXTENDS L_MC1P_AxisExtensionEmpty
VAR
	CONFIGDRIVE : L_MC1P_Config_GenericDrive;
	DRIVESCALING : L_MC1P_DriveScaling_GenericDrive;
	DRIVESPECIFIC : L_MC1P_DriveSpecific_Generic;
	ECATCOMM : L_MC1P_CommECAT;
	FBEXTENDEDMAPPINGACCESS : L_MC1P_ExtendedMappingAccess;
	GETTYPE : L_MC1P_AxisExtensionTypes;
	ITFCOMM : L_MC1P_ICommunication;
	ITFCONFIGDRIVE : L_MC1P_IConfigureDrive;
	ITFDRIVESCALING : L_MC1P_IDriveScaling;
	ITFDRIVESPECIFIC : L_MC1P_IDriveSpecificImplBase;
	ITFEXTENDEDMAPPINGACCESS : L_MC1P_IExtendedMappingAccess;
END_VAR
END_FUNCTION_BLOCK

METHOD SETBASICINITIALISATION
VAR_INPUT
	ITFGENERICCONFIG : L_MC1P_IGenericAxisConfiguration;
END_VAR
VAR_IN_OUT
	AXIS : _AXIS_REF_REAL;
END_VAR
END_METHOD

(* ---- L_MC1P_AXISEXTENSION_I500_CAN.pou ---- *)
FUNCTION_BLOCK L_MC1P_AXISEXTENSION_I500_CAN EXTENDS L_MC1P_AxisExtensionEmpty
VAR_INPUT
	DRIVESPECIFIC : L_MC1P_DriveSpecific_i500;
END_VAR
VAR
	CONFIGDRIVE : L_MC1P_Config_i500;
	DRIVESCALING : L_MC1P_DriveScaling_i500;
	CANCOMM : L_MC1P_CommCAN;
	ITFCOMM : L_MC1P_ICommunication;
	ITFCONFIGDRIVE : L_MC1P_IConfigureDrive;
	ITFDRIVESCALING : L_MC1P_IDriveScaling;
	ITFDRIVESPECIFIC : L_MC1P_IDriveSpecificImplBase;
END_VAR
END_FUNCTION_BLOCK

METHOD FB_INIT : BOOL
VAR_INPUT
	BINITRETAINS : BOOL;
	BINCOPYCODE : BOOL;
END_VAR
END_METHOD

(* ---- L_MC1P_AXISEXTENSION_I500_ECAT.pou ---- *)
FUNCTION_BLOCK L_MC1P_AXISEXTENSION_I500_ECAT EXTENDS L_MC1P_AxisExtensionEmpty
VAR_INPUT
	DRIVESPECIFIC : L_MC1P_DriveSpecific_i500;
END_VAR
VAR
	CONFIGDRIVE : L_MC1P_Config_i500;
	DRIVESCALING : L_MC1P_DriveScaling_i500;
	ECATCOMM : L_MC1P_CommECAT;
	FBEXTENDEDMAPPINGACCESS : L_MC1P_ExtendedMappingAccess;
	ITFCOMM : L_MC1P_ICommunication;
	ITFCONFIGDRIVE : L_MC1P_IConfigureDrive;
	ITFDRIVESCALING : L_MC1P_IDriveScaling;
	ITFDRIVESPECIFIC : L_MC1P_IDriveSpecificImplBase;
	ITFEXTENDEDMAPPINGACCESS : L_MC1P_IExtendedMappingAccess;
END_VAR
END_FUNCTION_BLOCK

(* ---- L_MC1P_AXISEXTENSION_I700.pou ---- *)
FUNCTION_BLOCK L_MC1P_AXISEXTENSION_I700 EXTENDS L_MC1P_AxisExtensionEmpty
VAR
	CONFIGDRIVE : L_MC1P_Config_i700_ETC;
	ECATCOMM : L_MC1P_CommECAT;
	FBEXTENDEDMAPPINGACCESS : L_MC1P_ExtendedMappingAccess;
	DRIVESCALING : L_MC1P_DriveScaling_i7xx;
	BRAKE : L_MC1P_BrakeControl;
	DRIVESPECIFIC : L_MC1P_DriveSpecific_i700;
	ITFCOMM : L_MC1P_ICommunication;
	ITFCONFIGDRIVE : L_MC1P_IConfigureDrive;
	ITFDRIVESCALING : L_MC1P_IDriveScaling;
	ITFDRIVESPECIFIC : L_MC1P_IDriveSpecificImplBase;
	ITFEXTENDEDMAPPINGACCESS : L_MC1P_IExtendedMappingAccess;
END_VAR
END_FUNCTION_BLOCK

METHOD FB_INIT : BOOL
VAR_INPUT
	BINITRETAINS : BOOL;
	BINCOPYCODE : BOOL;
END_VAR
END_METHOD

(* ---- L_MC1P_AXISEXTENSION_I750.pou ---- *)
FUNCTION_BLOCK L_MC1P_AXISEXTENSION_I750 EXTENDS L_MC1P_AxisExtensionEmpty
VAR
	CONFIGDRIVE : L_MC1P_Config_i900Adv_ETC;
	ECATCOMM : L_MC1P_CommECAT;
	FBEXTENDEDMAPPINGACCESS : L_MC1P_ExtendedMappingAccess;
	DRIVESCALING : L_MC1P_DriveScaling_i7xx;
	BRAKE : L_MC1P_BrakeControl;
	DRIVESPECIFIC : L_MC1P_DriveSpecific_i750;
	ITFCOMM : L_MC1P_ICommunication;
	ITFCONFIGDRIVE : L_MC1P_IConfigureDrive;
	ITFDRIVESCALING : L_MC1P_IDriveScaling;
	ITFDRIVESPECIFIC : L_MC1P_IDriveSpecificImplBase;
	ITFEXTENDEDMAPPINGACCESS : L_MC1P_IExtendedMappingAccess;
END_VAR
END_FUNCTION_BLOCK

METHOD FB_INIT : BOOL
VAR_INPUT
	BINITRETAINS : BOOL;
	BINCOPYCODE : BOOL;
END_VAR
END_METHOD

(* ---- L_MC1P_AXISEXTENSION_I950.pou ---- *)
FUNCTION_BLOCK L_MC1P_AXISEXTENSION_I950 EXTENDS L_MC1P_AxisExtensionEmpty
VAR
	CONFIGDRIVE : L_MC1P_Config_i900Adv_ETC := STRUCT(xCiA402Advanced := FALSE);
	ECATCOMM : L_MC1P_CommECAT;
	FBEXTENDEDMAPPINGACCESS : L_MC1P_ExtendedMappingAccess;
	BRAKE : L_MC1P_BrakeControl;
	DRIVESCALING : L_MC1P_DriveScaling_i7xx;
	DRIVESPECIFIC : L_MC1P_DriveSpecific_i950;
	ITFCOMM : L_MC1P_ICommunication;
	ITFCONFIGDRIVE : L_MC1P_IConfigureDrive;
	ITFDRIVESCALING : L_MC1P_IDriveScaling;
	ITFDRIVESPECIFIC : L_MC1P_IDriveSpecificImplBase;
	ITFEXTENDEDMAPPINGACCESS : L_MC1P_IExtendedMappingAccess;
END_VAR
END_FUNCTION_BLOCK

METHOD FB_INIT : BOOL
VAR_INPUT
	BINITRETAINS : BOOL;
	BINCOPYCODE : BOOL;
END_VAR
END_METHOD

(* ---- L_MC1P_AXISEXTENSION_I950_CIAADV.pou ---- *)
FUNCTION_BLOCK L_MC1P_AXISEXTENSION_I950_CIAADV EXTENDS L_MC1P_AxisExtensionEmpty
VAR
	CONFIGDRIVE : L_MC1P_Config_i900Adv_ETC := STRUCT(xCiA402Advanced := TRUE);
	ECATCOMM : L_MC1P_CommECAT;
	FBEXTENDEDMAPPINGACCESS : L_MC1P_ExtendedMappingAccess;
	DRIVESCALING : L_MC1P_DriveScaling_i7xx;
	BRAKE : L_MC1P_BrakeControl;
	DRIVESPECIFIC : L_MC1P_DriveSpecific_i950Adv;
	ITFCOMM : L_MC1P_ICommunication;
	ITFCONFIGDRIVE : L_MC1P_IConfigureDrive;
	ITFDRIVESCALING : L_MC1P_IDriveScaling;
	ITFDRIVESPECIFIC : L_MC1P_IDriveSpecificImplBase;
	ITFEXTENDEDMAPPINGACCESS : L_MC1P_IExtendedMappingAccess;
END_VAR
END_FUNCTION_BLOCK

METHOD FB_INIT : BOOL
VAR_INPUT
	BINITRETAINS : BOOL;
	BINCOPYCODE : BOOL;
END_VAR
END_METHOD

(* ---- L_MC1P_AXISEXTENSION_I950_DRIVE.pou ---- *)
FUNCTION_BLOCK L_MC1P_AXISEXTENSION_I950_DRIVE EXTENDS L_MC1P_AxisExtensionEmpty
VAR_INPUT
	CONFIGDRIVE : L_MC1P_Config_i900_Drive;
	COMM : L_MC1P_Commi900;
END_VAR
VAR
	DRIVESCALING : L_MC1P_DriveScaling_i7xx;
	BRAKE : L_MC1P_BrakeControlBase;
	DRIVESPECIFIC : L_MC1P_DriveSpecific_i950_Drive;
	ITFCOMM : L_MC1P_ICommunication;
	ITFCONFIGDRIVE : L_MC1P_IConfigureDrive;
	ITFDRIVESCALING : L_MC1P_IDriveScaling;
	ITFDRIVESPECIFIC : L_MC1P_IDriveSpecificImplBase;
END_VAR
END_FUNCTION_BLOCK

METHOD FB_INIT : BOOL
VAR_INPUT
	BINITRETAINS : BOOL;
	BINCOPYCODE : BOOL;
END_VAR
END_METHOD

(* ---- L_MC1P_AXISEXTENSIONEMPTY.pou ---- *)
FUNCTION_BLOCK L_MC1P_AXISEXTENSIONEMPTY
VAR
	GETTYPE : L_MC1P_AxisExtensionTypes;
	ITFCOMM : L_MC1P_ICommunication;
	ITFCONFIGDRIVE : L_MC1P_IConfigureDrive;
	ITFDRIVESCALING : L_MC1P_IDriveScaling;
	ITFDRIVESPECIFIC : L_MC1P_IDriveSpecificImplBase;
	ITFEXTENDEDMAPPINGACCESS : L_MC1P_IExtendedMappingAccess;
END_VAR
END_FUNCTION_BLOCK

METHOD SETBASICINITIALISATION
VAR_INPUT
	ITFGENERICCONFIG : L_MC1P_IGenericAxisConfiguration;
END_VAR
VAR_IN_OUT
	AXIS : _AXIS_REF_REAL;
END_VAR
END_METHOD

METHOD FB_EXIT : BOOL
VAR_INPUT
	BINCOPYCODE : BOOL;
END_VAR
END_METHOD

(* ---- L_MC1P_AXISINTERFACE.pou ---- *)
FUNCTION_BLOCK L_MC1P_AXISINTERFACE EXTENDS L_MC1P_Template
VAR_INPUT
	XENABLE : BOOL;
	EXTCONTROLLER : L_MC1P_IControllerInterface;
END_VAR
VAR_OUTPUT
	XVALID : BOOL;
	XBUSY : BOOL;
	XERROR : BOOL;
	EERRORID : L_IE1P_Error;
END_VAR
VAR
	XENABLEOLD : BOOL;
END_VAR
END_FUNCTION_BLOCK

(* ---- L_MC1P_AXISMANAGEMENTFUNCTION.pou ---- *)
FUNCTION_BLOCK L_MC1P_AXISMANAGEMENTFUNCTION
VAR
	LMAXISMANAGEMENTFUNCTION : ARRAY [1..L_MC1P_Constants.gc_MaxAxisCount] OF L_MC1P_IManagementFunction;
	DIAXISCOUNT : DINT;
END_VAR
END_FUNCTION_BLOCK

METHOD FINDAXISBYNAME : POINTER TO AXIS_REF
VAR_IN_OUT
	SAXISNAME : STRING;
END_VAR
END_METHOD

METHOD GETFIRSTAXIS : POINTER TO AXIS_REF
VAR_INPUT
	PIDX : POINTER TO DINT;
END_VAR
END_METHOD

METHOD GETNEXTAXIS : POINTER TO AXIS_REF
VAR_INPUT
	PIDX : POINTER TO DINT;
END_VAR
END_METHOD

METHOD REGISTERAXIS : BOOL
VAR_INPUT
	ITFMANAGE : L_MC1P_IManagementFunction;
END_VAR
END_METHOD

(* ---- L_MC1P_AXISMASTERVALUESEMPTY.pou ---- *)
FUNCTION_BLOCK L_MC1P_AXISMASTERVALUESEMPTY
VAR
	FBSTEADYSTATE : L_MC1P_SteadyState;
	ACTACCELERATION : LREAL;
	ACTPOSITION : LREAL;
	ACTTORQUE : LREAL;
	ACTVELOCITY : LREAL;
	CYCLELENGTH : LREAL;
	FEEDCONSTANT : LREAL;
	GETMASTERID : POINTER TO BYTE;
	SETACCELERATIONFORSYNC : LREAL;
	SETPOSITIONFORSYNC : LREAL;
	SETTORQUEFORSYNC : LREAL;
	SETVELOCITYFORSYNC : LREAL;
	TASKCYCLE : LREAL;
	TRAVERSINGRANGE : L_MC1P_TraversingRange;
END_VAR
END_FUNCTION_BLOCK

METHOD GETDIRECTION : WORD
VAR_INPUT
	VALUESOURCE : MC_SOURCE;
END_VAR
END_METHOD

METHOD GETMASTERERROR : BOOL
VAR_OUTPUT
	EERRORID : L_IE1P_Error;
END_VAR
END_METHOD

METHOD GETSTEADYSTATE : POINTER TO L_MC1P_SteadyState
END_METHOD

(* ---- L_MC1P_AXISRETAINMANGAEMENT.pou ---- *)
FUNCTION_BLOCK L_MC1P_AXISRETAINMANGAEMENT
VAR_OUTPUT
	XERROR : BOOL;
END_VAR
VAR
	XINIT : BOOL := FALSE;
	ERRORHANDLE : SysTypes.RTS_IEC_HANDLE := 0;
	MODULEHANDLE : SysTypes.RTS_IEC_HANDLE := 0;
	DWLENGTH : DWORD;
	XMEMVALID : BOOL := FALSE;
	PSTARTADRESS : POINTER TO DWORD;
	PMEMADRESS : POINTER TO DWORD;
	PMEMADRESSMIRROR : POINTER TO DWORD;
	DWMEMSIZE : DWORD;
	DIAXISCOUNT : DINT := 0;
	LMAXISINFORMATION : ARRAY [1..L_MC1P_Constants.gc_MaxRetainAxis] OF L_MC1P_AxisRetainInformation;
	WSTEP : WORD := 0;
	XCONFIGCHANGED : BOOL;
	DATAMEMORYAREA : L_SSYP_PersistantDataMemoryArea;
	DWVERSION : DWORD;
	XINITIALAREA : BOOL := FALSE;
	DWTOTALSIZE1 : DWORD;
	DWTOTALSIZE2 : DWORD;
	PADWDUMMY1 : POINTER TO ARRAY [1..100] OF DWORD;
	PADWDUMMY2 : POINTER TO ARRAY [1..100] OF DWORD;
	WINTSTATE : WORD;
	DIIDX : DINT;
	BYMEMVERSION : BYTE;
	SINSTANCESTRFULL : STRING(255);
	BYACTMEMVERSION : BYTE := 2;
END_VAR
END_FUNCTION_BLOCK

METHOD CHECKMEMORY
END_METHOD

METHOD GETDATA : BOOL
VAR_IN_OUT
	AXISRETAIN : L_MC1P_AxisRetainInformation;
END_VAR
END_METHOD

METHOD READDWORD : DWORD
VAR_IN_OUT
	DWSIZEREAD : DWORD;
END_VAR
END_METHOD

METHOD READMEMORY
END_METHOD

METHOD REINITMEMORY
VAR_INPUT
	PDATA : POINTER TO DWORD;
	XMIRROR : BOOL;
END_VAR
END_METHOD

METHOD SEARCHDATA : BOOL
VAR_IN_OUT
	DWSIZEREAD : DWORD;
	AXISRETAIN : L_MC1P_AxisRetainInformation;
END_VAR
END_METHOD

METHOD SETACTIVEMEMAREA
VAR_INPUT
	XMIRROR : BOOL;
END_VAR
END_METHOD

METHOD SETMEMORYINVALID
END_METHOD

METHOD WRITEAXISDATA
END_METHOD

METHOD WRITEDWORD : DWORD
VAR_INPUT
	PMEMBASE : POINTER TO DWORD;
	DWDATA : DWORD;
END_VAR
VAR_IN_OUT
	DWSIZEWRITE : DWORD;
END_VAR
END_METHOD

METHOD FB_EXIT : BOOL
VAR_INPUT
	BINCOPYCODE : BOOL;
END_VAR
END_METHOD

METHOD FB_INIT : BOOL
VAR_INPUT
	BINITRETAINS : BOOL;
	BINCOPYCODE : BOOL;
END_VAR
END_METHOD

METHOD REGISTERAXIS
VAR_INPUT
	AXISGUID : L_MC1P_AxisGUID;
END_VAR
END_METHOD

METHOD REGISTERAXIS2 : POINTER TO L_MC1P_AxisRetainInformation
VAR_INPUT
	AXISGUID : L_MC1P_AxisGUID;
	ITFRETAIN : L_MC1P_IRetainFunction;
END_VAR
END_METHOD

METHOD INITMEMFORAXIS
VAR_INPUT
	PDATA : POINTER TO DWORD;
	XMIRROR : BOOL;
END_VAR
VAR_IN_OUT
	DWWRITEOFFSET : DWORD;
	AXISRETAININFORMATION : L_MC1P_AxisRetainInformation;
END_VAR
END_METHOD

METHOD WRITEADDSIZE
VAR_INPUT
	PDATA : POINTER TO DWORD;
	DWADDSIZE : DWORD;
END_VAR
END_METHOD

METHOD WRITEHEADER
VAR_INPUT
	PDATA : POINTER TO DWORD;
END_VAR
END_METHOD

(* ---- L_MC1P_AXISSIMREADPRM.pou ---- *)
FUNCTION_BLOCK L_MC1P_AXISSIMREADPRM EXTENDS L_UBUP_FreeRunTask
VAR_INPUT
	UIDEVICEID : UINT;
	PPARAMDATA : POINTER TO L_MC1P_ParameterDataSim;
	WPARAMCOUNT : WORD;
	PPARAMDATAIGNORE : POINTER TO L_MC1P_ParameterDataSim;
	WPARAMCOUNTIGNORE : WORD;
END_VAR
VAR
	PARSIMWRITE : L_MC1P_ParSimWrite;
	SBASEPATH : STRING(255);
END_VAR
END_FUNCTION_BLOCK

METHOD CUSTOMIZEERRORCODE : L_IE1P_Error
VAR_INPUT
	IERRORID : INT;
END_VAR
END_METHOD

METHOD EXECUTEIMPL : UDINT
END_METHOD

METHOD FB_INIT : BOOL
VAR_INPUT
	BINITRETAINS : BOOL;
	BINCOPYCODE : BOOL;
END_VAR
END_METHOD

(* ---- L_MC1P_AXISSIMULATION.pou ---- *)
FUNCTION_BLOCK L_MC1P_AXISSIMULATION
VAR_INPUT
	SCIODATA : L_MC1P_AxisSimIOData;
	SCPARMECHANIC : L_MC1P_ParMechanic;
	SCPAROBDDRIVE : L_MC1P_AxisSimulationSdoData;
	SCPARGENERAL : L_MC1P_ParGeneralMechanic;
	LRINITIALPOSITION : LREAL;
	EINITOBDDRIVEMODE : UINT := 0;
END_VAR
VAR_OUTPUT
	XBUSY : BOOL;
END_VAR
VAR
	COMMUNICATION : L_MC1P_CommSim;
	APARAMDATA : ARRAY [1..c_MaxSimData] OF L_MC1P_ParameterDataSim;
	APRMIGNOREDATA : ARRAY [1..c_MaxPrmIgnoreData] OF L_MC1P_ParameterDataSim;
	TRANSMITDATA : L_MC1P_AxisSimulationPDOdataToDrive;
	RECIEVEDATA : L_MC1P_AxisSimulationPDOdataFromDrive;
	LWTRANSDATA : LWORD;
	LWTRANSDATASAVE : LWORD;
	WTRANSELEMENTS : WORD;
	ATRANSELEMENT : ARRAY [1..c_wMaxTransElem] OF L_MC1P_MappedElement;
	ATRANSELEMENTADRESS : ARRAY [1..L_MC1P_Constants.gc_Trans_MaxDataIndex] OF POINTER TO L_MC1P_MappedElement;
	ATRANSELEMENTADRESSSAVE : ARRAY [1..L_MC1P_Constants.gc_Trans_MaxDataIndex] OF POINTER TO L_MC1P_MappedElement;
	LWRECDATA : LWORD;
	LWRECDATASAVE : LWORD;
	WRECEIVEELEMENTS : WORD;
	ARECEIVEELEMENT : ARRAY [1..c_wMaxRecElem] OF L_MC1P_MappedElement;
	ARECEIVEELEMENTADRESS : ARRAY [1..L_MC1P_Constants.gc_Rec_MaxDataIndex] OF POINTER TO L_MC1P_MappedElement;
	ARECEIVEELEMENTADRESSSAVE : ARRAY [1..L_MC1P_Constants.gc_Rec_MaxDataIndex] OF POINTER TO L_MC1P_MappedElement;
	IBUSDEADCYCLES : INT := 2;
	IINDEXPDO : INT := 1;
	ASCPDO_P2D : ARRAY [0..(ciPDO_BufferSize - 1)] OF L_MC1P_AxisSimulationPDOdataToDrive;
	ASCPDO_D2P : ARRAY [0..(ciPDO_BufferSize - 1)] OF L_MC1P_AxisSimulationPDOdataFromDrive;
	SYSTEMSIMULATION : L_MC1P_SimMotorCtrl;
	MECHANICSIMULATION : L_MC1P_SimMechanic;
	ITFMECHANICMODELDEFAULT : L_MC1P_IMechanicSimulation := MechanicSimulation;
	ITFMECHANICMODELACT : L_MC1P_IMechanicSimulation := itfMechanicModelDefault;
	TRANSMITDATASCALED : L_MC1P_AxisSimulationPDOdataToDriveScaled;
	RECIEVEDATASCALED : L_MC1P_AxisSimulationPDOdataFromDriveScaled;
	XREADPARSET : BOOL;
	AXISSIMREADPRM : L_MC1P_AxisSimReadPRM;
	XGENERRORREAKTINDEVICESAVE : BOOL;
	C_WMAXTRANSELEM : WORD := 20;
	C_WMAXRECELEM : WORD := 38;
	C_MAXSIMDATA : WORD := 90;
	C_MAXPRMIGNOREDATA : WORD := 5;
	CIPDO_BUFFERSIZE : INT := 10;
	COMMSIMULATION : L_MC1P_ICommmunicationSimulation;
	GETRECIEVEDATACONFIG : LWORD;
	GETTRANSMITDATACONFIG : LWORD;
	LOADFDB : LREAL;
	RECIEVEELEMCOUNT : WORD;
	RECIEVEELEMENT : POINTER TO L_MC1P_MappedElement;
	RECIEVEELEMENTADRESS : POINTER TO ARRAY [1..L_MC1P_Constants.gc_Rec_MaxDataIndex] OF POINTER TO L_MC1P_MappedElement;
	TRANSELEMCOUNT : WORD;
	TRANSELEMENT : POINTER TO L_MC1P_MappedElement;
	TRANSELEMENTADRESS : POINTER TO ARRAY [1..L_MC1P_Constants.gc_Trans_MaxDataIndex] OF POINTER TO L_MC1P_MappedElement;
END_VAR
END_FUNCTION_BLOCK

METHOD SETMECHANICMODEL : BOOL
VAR_INPUT
	ITFMECHANICMODEL : L_MC1P_IMechanicSimulation;
END_VAR
END_METHOD

METHOD CALCOPTIMIZEDMAPPINGINFO : BOOL
END_METHOD

METHOD GETBITNBR : WORD
VAR_INPUT
	LWMASK : LWORD;
END_VAR
END_METHOD

METHOD INITOBD : BOOL
END_METHOD

METHOD SETDRIVEDEPENDENTMAPPING : BOOL
VAR_IN_OUT
	AXIS : _AXIS_REF_REAL;
END_VAR
END_METHOD

METHOD SETPARAMETERINFO : BOOL
VAR_INPUT
	PARAMDATAIDX : WORD;
	WINDEX : WORD;
	BYSUBINDEX : BYTE;
	PDOMAPNBR : LWORD;
	PDATA : POINTER TO BYTE;
	BYNROFBYTE : BYTE;
	XSUPPORTED : BOOL;
	XWRITEACCESS : BOOL;
	XAXISOFFSET : BOOL;
	EFIXTOLREAL : L_MC1P_ScaleFixToLREAL := L_MC1P_ScaleFixToLREAL.None;
END_VAR
END_METHOD

METHOD FB_INIT : BOOL
VAR_INPUT
	BINITRETAINS : BOOL;
	BINCOPYCODE : BOOL;
END_VAR
END_METHOD

METHOD GETBUSVALUESP2D
VAR_IN_OUT
	AXIS : _AXIS_REF_REAL;
END_VAR
END_METHOD

METHOD WRITEBUSVALUESD2P
VAR_IN_OUT
	AXIS : _AXIS_REF_REAL;
END_VAR
END_METHOD

METHOD ACTIVATESIMULATION
VAR_IN_OUT
	AXIS : _AXIS_REF_REAL;
END_VAR
END_METHOD

METHOD CALCULATEINPUTDATA
VAR_IN_OUT
	AXIS : _AXIS_REF_REAL;
END_VAR
END_METHOD

METHOD CALCULATEOUTPUTDATA
VAR_IN_OUT
	AXIS : _AXIS_REF_REAL;
END_VAR
END_METHOD

METHOD DISABLESIMULATION
VAR_IN_OUT
	AXIS : _AXIS_REF_REAL;
END_VAR
END_METHOD

(* ---- L_MC1P_BASICACTUATINGSPEED.pou ---- *)
FUNCTION_BLOCK L_MC1P_BASICACTUATINGSPEED EXTENDS L_MC1P_Template
VAR_INPUT
	XENABLEINTERNALCONTROL : BOOL := FALSE;
	XREGULATORON : BOOL := FALSE;
	XRESETERROR : BOOL := FALSE;
	XSETDRIVEQSP : BOOL := FALSE;
	XENABLESETVEL : BOOL := FALSE;
	XINVERTDIRECTION : BOOL := FALSE;
	LRSETVEL : LREAL := 0.0;
	LRSETACC : LREAL := 0.0;
	LRSETDEC : LREAL := 0.0;
END_VAR
VAR_OUTPUT
	XINTERNALCONTROLACTIVE : BOOL;
	XBUSY : BOOL;
	XERROR : BOOL;
	EERRORID : L_IE1P_Error;
	XCOMMUNICATIONOK : BOOL;
	XAXISREADY : BOOL;
	XAXISENABLED : BOOL;
	XDRIVEWARNING : BOOL;
	XDRIVEERROR : BOOL;
	DWDRIVEERRORID : DWORD;
	XDRIVEQSPACTIVE : BOOL;
	LRACTVEL : LREAL;
	XDIRECTIONPOSITIVE : BOOL;
	XDIRECTIONNEGATIVE : BOOL;
	WDIGITALINPUTS : WORD;
END_VAR
VAR
	XINTERNALCONTROLVISU : BOOL;
	XREGULATORON_INT : BOOL := FALSE;
	XSETDRIVEQSP_INT : BOOL := FALSE;
	XRESETERROR_INT : BOOL := FALSE;
	XENABLESETVEL_INT : BOOL := FALSE;
	XINVERTDIRECTION_INT : BOOL := FALSE;
	LRSETVEL_INT : LREAL := 0.0;
	LRSETACC_INT : LREAL := 0.0;
	LRSETDEC_INT : LREAL := 0.0;
	LRSETACCOLD : LREAL := 0.0;
	LRSETDECOLD : LREAL := 0.0;
	LRSCALERPMTOUNITOLD : LREAL := 0.0;
	READAXISERROR : L_MC1P_ReadAxisError_Internal;
	FBRESET : L_MC1P_Reset_Internal;
	DWDIGIN : DWORD;
	PREALAXIS : POINTER TO _AXIS_REF_REAL;
	PWDUMMY : POINTER TO WORD;
	PXDUMMY : POINTER TO BOOL;
	BYSDORETRYCOUNTER : BYTE;
	XWAITFORPARAMETERWRITEDONE : BOOL;
	WRITEPARAMETER : L_DCO_WriteDriveParameter;
	WSTEP : WORD;
	DWDELTASPEED : DWORD;
	WDELTATIME : WORD;
	XINTERNALCONTROLACTIVEOLD : BOOL;
	WLCONTROLWORD : WORD;
	WLCONTROLWORD2 : WORD;
	WLCONTROLWORD3 : WORD;
	WLCONTROLWORD4 : WORD;
	WLSTATUSWORD : WORD;
	WLSTATUSWORD2 : WORD;
	PITFMANIPULATEACTVALUES : POINTER TO L_Mc1P_IManipulateActValues;
	MAX_SDO_RETRIES : WORD := 3;
	LCONTROLWORD : WORD;
	LCONTROLWORD2 : WORD;
	LCONTROLWORD3 : WORD;
	LCONTROLWORD4 : WORD;
	LSTATUSWORD : WORD;
	LSTATUSWORD2 : WORD;
END_VAR
END_FUNCTION_BLOCK

METHOD CALCACCVALUES
VAR_INPUT
	LRACC : LREAL;
END_VAR
VAR_OUTPUT
	DWDELTASPEED : DWORD;
	WDELTATIME : WORD;
END_VAR
VAR_IN_OUT
	REALAXIS : _AXIS_REF_REAL;
END_VAR
END_METHOD

METHOD CHECKACCDECCHANGED
VAR_IN_OUT
	REALAXIS : _AXIS_REF_REAL;
END_VAR
END_METHOD

METHOD MANIPULATEACTVALUES
VAR_IN_OUT
	AXIS : AXIS_REF;
END_VAR
END_METHOD

(* ---- L_MC1P_BRAKECONTROL.pou ---- *)
FUNCTION_BLOCK L_MC1P_BRAKECONTROL EXTENDS L_MC1P_BrakeControlBase
VAR_INPUT
	LRTORQUEADD : LREAL;
	XSTARTINGTORQUE2 : BOOL;
	LRBRAKERAMPTIME : REFERENCE TO LREAL;
	XBRAKEACCDEPENDING : REFERENCE TO BOOL;
	LRSPEEDMIN : LREAL;
	LRRAMPWATCHTIME : LREAL;
	WSOURCESTARTVALUE : REFERENCE TO WORD;
	ALRMSTARTVALUE : REFERENCE TO ARRAY [1..2] OF LREAL;
	LREFFECTIVESTARTINGTORQUE : REFERENCE TO LREAL;
END_VAR
VAR
	LRSPEEDSET : LREAL;
	LRSPEEDACT : LREAL;
	XMOTORPHASESOK : BOOL := TRUE;
	MCTRLCONF : L_MC1P_MctrlControl := L_MC1P_MctrlControl.mcStandard;
	XESSACTIVE : BOOL := FALSE;
	XFLYINGSYNCBUSY : BOOL;
	XDCBRAKEISACTIVE : BOOL := FALSE;
	XDCBRAKEINSTEADQSP : BOOL := FALSE;
	XQSPISACTIVE : BOOL := FALSE;
	XSLIPCTRLACTIVE : BOOL := FALSE;
	XMAGNETISATIONISFINISHED : BOOL := FALSE;
	XUVDETECTED : BOOL;
	LRMAGNETISATIONTIME : LREAL := 1.0;
	LRTASKCYCLE : LREAL := 0.001;
	LRREFERENCETORQUE : LREAL;
	XINVERTBRAKECTRL : BOOL;
	XBRAKESTATEINPUT : BOOL;
	XIMPBRAKEREACTION : BOOL;
	LRBRAKEOBSERVATIONDELAY : LREAL;
	XBRAKEFEEDBACK : BOOL;
	XGETCINH_NOBRAKE : BOOL;
	XBRKSETCINH : BOOL;
	LRSETSPEEDOUT : LREAL;
	XBRAKEAPPLIED : BOOL;
	LRTORQUESET : LREAL;
	LRSPEEDSETOLD : LREAL;
	LRSPEEDACTOLD : LREAL;
	LRSPEEDCTRLINTVALUESET : LREAL;
	XLASTSPEEDBELOWMINSPEED : BOOL;
	LRTIMEOUTCOUNTER : LREAL;
	LRRELEASECOUNTER : LREAL;
	LROBSERVATIONCOUNTER : LREAL;
	XAUTOSUPERVISOROLD : BOOL;
	LRTORQUEACTFILTERED : LREAL;
	XSPEEDEQZERO : BOOL;
	XAXISERROR : BOOL;
	XQSPACTIVE : BOOL;
	XSETSPEEDTOZERO : BOOL;
	XAXISCINH : BOOL;
	LRAXISDECERRSTOP : LREAL;
	LRAXISJERKERRSTOP : LREAL;
	XBRAKEMODEINIT : BOOL;
	LRDRIVEMODEOBERSERVATIONCOUNTER : LREAL;
	XCIASTATUS : BOOL;
	DIPOSACT2NDSOURCE : DINT;
	DIBRAKEPOSITION2NDSOURCE : DINT;
	X2NDPOSVALID : BOOL;
	READPOS2NDSOURCE : L_DCO_ReadDriveParameter;
	XACTIVATEBRAKEMODEOBSERVATION : BOOL := TRUE;
	XDELAYOPERATIONENABLEDINACTIVE : BOOL := TRUE;
	XCLOSEBRAKEBECAUSOFFAULTREACTION : BOOL := FALSE;
	XCLOSEBRAKEATQSPRAMPEND : BOOL := FALSE;
	BRAKELOGICINPLCACTIVE : BOOL;
	PINSTANCE : POINTER TO L_MC1P_BrakeControlBase;
	TORQUEPRECONTROLACTIVE : BOOL;
END_VAR
END_FUNCTION_BLOCK

METHOD BF_BRAKE
END_METHOD

METHOD CONNECTPARAMETER : BOOL
VAR_INPUT
	PBRAKEPARA : POINTER TO L_MC1P_BrakePara;
END_VAR
END_METHOD

METHOD INIT
VAR_INPUT
	WBRAKEMODEINDEXOFDRIVE : WORD;
	BYSUBINDEX : BYTE;
	SZSIZE : BYTE;
	DEFAULTVALUE : DWORD;
END_VAR
VAR_IN_OUT
	AXIS : AXIS_REF;
END_VAR
END_METHOD

METHOD SUPPORTEDFUNCTION : INT
END_METHOD

METHOD FB_INIT : BOOL
VAR_INPUT
	BINITRETAINS : BOOL;
	BINCOPYCODE : BOOL;
END_VAR
END_METHOD

METHOD MODEAUTOENTERBRAKECLOSED
END_METHOD

METHOD MODEAUTOSTATEBRAKECLOSED
END_METHOD

METHOD MODEAUTOENTERCLOSINGBRAKE
END_METHOD

METHOD MODEAUTOENTERRAMPDOWN
END_METHOD

METHOD MODEAUTOSTATECLOSINGBRAKE
END_METHOD

METHOD MODEAUTOSTATERAMPDOWN
END_METHOD

METHOD BRAKECLEARERROR
VAR_INPUT
	ERRORCODE : L_MC1P_BrakeErrorCodes;
END_VAR
END_METHOD

METHOD BRAKERAISEERROR
VAR_INPUT
	ERRORCODE : L_MC1P_BrakeErrorCodes;
END_VAR
END_METHOD

METHOD ACTSPEEDISBELOWMINSPEED : BOOL
END_METHOD

METHOD BF_BRAKECLOSE
END_METHOD

METHOD BF_BRAKEDIRECTMODE
VAR_INPUT
	XSETDIRECTMODE : BOOL;
END_VAR
END_METHOD

METHOD BF_BRAKEGETSTATE : L_MC1P_BrakeState
VAR_OUTPUT
	ESTATEOPERATION : INT;
END_VAR
END_METHOD

METHOD BF_BRAKEGETSTATE_STATECONTROL : L_MC1P_BrakeState
END_METHOD

METHOD BF_BRAKEOPEN
END_METHOD

METHOD BF_BRAKEOUTPUTS
END_METHOD

METHOD BF_FQSPACTIVE : BOOL
END_METHOD

METHOD BF_TRIPACTIVE : BOOL
END_METHOD

METHOD BRAKEMODEOFF
END_METHOD

METHOD BRAKEMODEVALID : BOOL
VAR_INPUT
	BRAKEMODE : L_MC1P_BrakeMode;
END_VAR
END_METHOD

METHOD CONVERTBRAKEMODE : L_MC1P_InternalBrakeMode
VAR_INPUT
	EMODE : L_MC1P_BrakeMode;
END_VAR
END_METHOD

METHOD GETACTSPEEDISBELOWMINSPEED : BOOL
END_METHOD

METHOD INITTORQUEPRECONTROL
END_METHOD

METHOD ISBRAKECLOSEREQUESTED : BOOL
END_METHOD

METHOD ISBRAKERELEASEREQUESTED : BOOL
END_METHOD

METHOD ISNOFEEDBACK : BOOL
END_METHOD

METHOD ISNOIMPBECAUSEOFDCBRAKE : BOOL
END_METHOD

METHOD MODEAUTO
END_METHOD

METHOD MODEAUTOSTATESUPERVISOR
END_METHOD

METHOD MODEDIRECTCONTROL
END_METHOD

METHOD MODEMANUAL
END_METHOD

METHOD RESETOUTPUTSTATE
END_METHOD

METHOD SETSPEEDISBELOWMINSPEED : BOOL
END_METHOD

METHOD SPEEDEQ0 : BOOL
VAR_INPUT
	LRACTSPEED : LREAL;
	LRACTSPEEDOLD : LREAL;
END_VAR
END_METHOD

METHOD GETACTVALUES
END_METHOD

METHOD SWITCHONCONTROL
VAR_INPUT
	XSWITCHONREQUEST : BOOL;
END_VAR
VAR_OUTPUT
	XSWITCHON : BOOL;
END_VAR
VAR_IN_OUT
	AXIS : AXIS_REF;
END_VAR
END_METHOD

METHOD SWITCHEDONSTATUS
VAR_INPUT
	XSWITCHEDONREQUEST : BOOL;
END_VAR
VAR_OUTPUT
	XSWITCHEDON : BOOL;
END_VAR
VAR_IN_OUT
	AXIS : AXIS_REF;
END_VAR
END_METHOD

METHOD MODEAUTOENTERIDLE
END_METHOD

METHOD MODEAUTOSTATEIDLE
END_METHOD

METHOD BRAKEPRECONTROLWHILECLOSING
END_METHOD

METHOD BRAKETORQUECONTROL : BOOL
END_METHOD

METHOD GENERATETORQUEPRECONTROL
VAR_INPUT
	PLRACTVAL : POINTER TO LREAL;
	LRENDVAL : LREAL;
END_VAR
END_METHOD

METHOD MODEAUTOENTERRELEASINGBRAKE
END_METHOD

METHOD MODEAUTOSTATERELEASINGBRAKE
END_METHOD

(* ---- L_MC1P_BRAKECONTROLBASE.pou ---- *)
FUNCTION_BLOCK L_MC1P_BRAKECONTROLBASE
VAR_INPUT
	XRELEASEBRAKE : BOOL;
	XEXTBRAKEMODE : BOOL := FALSE;
	EEXTBRAKEMODE : L_MC1P_BrakeMode := L_MC1P_BrakeMode.Off;
	XEXTBRAKEMODESERVICE : BOOL := FALSE;
	EEXTBRAKEMODESERVICE : L_MC1P_BrakeMode := L_MC1P_BrakeMode.Off;
	DWBRAKEMODE : REFERENCE TO DWORD;
	LRRELEASETIME : REFERENCE TO LREAL;
	LRACTIVATIONTIME : REFERENCE TO LREAL;
	LRRELEASETIMEUSED : LREAL := 0.1;
	LRACTIVATIONTIMEUSED : LREAL := 0.1;
	XEXTBRAKETIMES : BOOL;
	LRRELEASETIMEEXT : LREAL := 0.1;
	LRACTIVATIONTIMEEXT : LREAL := 0.1;
	LRPOSFAILTHRESHOLDBRAKETEST : LREAL;
	XBRAKETEST : BOOL;
	LRSAMPLEDBRAKETORQUE : REFERENCE TO LREAL;
	LRPOSFAILTHRESHOLD : LREAL;
	XREAD2NDPOS : BOOL;
	LRDELTAPOS2NDSOURCE : LREAL;
	XRELEASEBRAKEALLOWEDINDIRECTMODE : BOOL;
	XENABLERELEASEBRAKEINAUTOMODE : BOOL := TRUE;
	XENABLERELEASEBRAKEINDIRECTMODE : BOOL;
	XTORQUETESTLIMITED : BOOL;
	XCLOSEBRAKESPEEDINDEPENDENT : BOOL;
	ESELBRAKEMODE : REFERENCE TO DWORD;
END_VAR
VAR_OUTPUT
	XRELEASEBRAKEOUTDISPLAY : BOOL;
	XRELEASEBRAKEOUT : BOOL;
	XBRAKERELEASED : BOOL;
	XERROR : BOOL;
	EERRORID : L_IE1P_Error;
END_VAR
VAR
	XIMPISACTIVE : BOOL;
	LRTORQUEACT : LREAL;
	XCINHISACTIVE : BOOL;
	PAXIS : POINTER TO _AXIS_REF_REAL;
	DIPOSACT : DINT;
	DIBRAKEPOSITION : DINT;
	XSTATUS : BOOL;
	XSWITCHONENABLED : BOOL;
	XBRAKEENABLED : BOOL := TRUE;
	XSETSPEEDCTRLINT : BOOL;
	XSETSPEEDCTRLINTOLD : BOOL;
	LRSPEEDCTRLINTVALUE : LREAL;
	ECURRENTSELBRAKEMODE : L_MC1P_BrakeMode := L_MC1P_BrakeMode.Off;
	SELECTEDBRAKEMODEINT : L_MC1P_InternalBrakeMode := L_MC1P_InternalBrakeMode.BM_Off;
	CURRENTBRAKEMODE : L_MC1P_InternalBrakeMode := L_MC1P_InternalBrakeMode.BM_Off;
	XERROROLD : BOOL;
	XBRAKEDIRECTMODE : BOOL;
	WP : L_DCO_WriteDriveParameter;
	WP_INIT : BOOL := FALSE;
	XWRITEBRAKEMODE : BOOL := FALSE;
	XWRITEBRAKEMODEDONE : BOOL;
	LRDELTAPOS : LREAL;
	BRAKECTRL : L_MC1P_BrakeCtrl;
	XOPENAUTOBRAKE : BOOL;
	XCLOSEAUTOBRAKE : BOOL;
	XTRIGGERCLOSEBRAKE : BOOL;
	BRAKEOVERRIDE : BYTE;
	DWLSTATEWORD2 : DWORD;
	DWCONTROLWORD : DWORD;
	XCONTROLWORDRELEASEBRAKEOUT : BOOL;
	XSTATEWORDBRAKERELEASED : BOOL;
	XCONTROLWORDRELEASEBRAKEOUT_OLD : BOOL;
	XSTATEWORDBRAKERELEASED_OLD : BOOL;
	MC_OVERRIDEBRAKECONTROL : MC_WriteParameter;
	OUTPUTSTATE : L_MC1P_BrakeOutState;
	EAUTOSTATE : L_MC1P_BrakeAutoState;
	XOUTPUTRELEASE : BOOL;
	XOUTPUTRELEASE_OLD : BOOL;
	XSPEEDFEEDBACK : BOOL := TRUE;
	DWACTIVEERRORS : DWORD;
	XOUTPUTERROR : BOOL;
	SCPARBRAKE : L_MC1P_BrakePara;
	BRAKELOGICINPLCACTIVE : BOOL;
	PINSTANCE : POINTER TO L_MC1P_BrakeControlBase;
	TORQUEPRECONTROLACTIVE : BOOL;
	TRIGGERCLOSEBRAKE : BOOL;
END_VAR
END_FUNCTION_BLOCK

METHOD BF_BRAKE
END_METHOD

METHOD CONNECTPARAMETER : BOOL
VAR_INPUT
	PBRAKEPARA : POINTER TO L_MC1P_BrakePara;
END_VAR
END_METHOD

METHOD INIT
VAR_INPUT
	WBRAKEMODEINDEXOFDRIVE : WORD;
	BYSUBINDEX : BYTE;
	SZSIZE : BYTE;
	DEFAULTVALUE : DWORD;
END_VAR
VAR_IN_OUT
	AXIS : AXIS_REF;
END_VAR
END_METHOD

METHOD SUPPORTEDFUNCTION : INT
END_METHOD

METHOD FB_INIT : BOOL
VAR_INPUT
	BINITRETAINS : BOOL;
	BINCOPYCODE : BOOL;
END_VAR
END_METHOD

METHOD BRAKECLEARERROR
VAR_INPUT
	ERRORCODE : L_MC1P_BrakeErrorCodes;
END_VAR
END_METHOD

METHOD BRAKERAISEERROR
VAR_INPUT
	ERRORCODE : L_MC1P_BrakeErrorCodes;
END_VAR
END_METHOD

METHOD BF_BRAKECLOSE
END_METHOD

METHOD BF_BRAKEDIRECTMODE
VAR_INPUT
	XSETDIRECTMODE : BOOL;
END_VAR
END_METHOD

METHOD BF_BRAKEGETSTATE : L_MC1P_BrakeState
VAR_OUTPUT
	ESTATEOPERATION : INT;
END_VAR
END_METHOD

METHOD BF_BRAKEGETSTATE_STATECONTROL : L_MC1P_BrakeState
END_METHOD

METHOD BF_BRAKEOPEN
END_METHOD

METHOD BRAKEMODEOFF
END_METHOD

METHOD BRAKEMODEVALID : BOOL
VAR_INPUT
	BRAKEMODE : L_MC1P_BrakeMode;
END_VAR
END_METHOD

METHOD ISBRAKERELEASEREQUESTED : BOOL
END_METHOD

METHOD MODEDIRECTCONTROL
END_METHOD

METHOD GETACTVALUES
END_METHOD

METHOD GETACTVALUESBRAKE
END_METHOD

METHOD SWITCHONCONTROL
VAR_INPUT
	XSWITCHONREQUEST : BOOL;
END_VAR
VAR_OUTPUT
	XSWITCHON : BOOL;
END_VAR
VAR_IN_OUT
	AXIS : AXIS_REF;
END_VAR
END_METHOD

METHOD SWITCHEDONSTATUS
VAR_INPUT
	XSWITCHEDONREQUEST : BOOL;
END_VAR
VAR_OUTPUT
	XSWITCHEDON : BOOL;
END_VAR
VAR_IN_OUT
	AXIS : AXIS_REF;
END_VAR
END_METHOD

(* ---- L_MC1P_BRAKEGRINDIN.pou ---- *)
FUNCTION_BLOCK L_MC1P_BRAKEGRINDIN EXTENDS L_MC1P_Template
VAR_INPUT
	XEXECUTE : BOOL;
	EMODE : L_MC1P_GrindInMode := L_MC1P_GrindInMode.CwCcw;
	EADDITIONALLIMITS : L_MC1P_AdditionalLimits := L_MC1P_AdditionalLimits.NotActive;
	LRPOSLIMIT1 : LREAL := 0;
	LRPOSLIMIT2 : LREAL := 0;
	LRMOTORSPEED : LREAL := 60.0;
	LRRAMPTIME : LREAL := 1.0;
	LRONTIME : LREAL := 0.5;
	LROFFTIME : LREAL := 0.5;
	WCYCLES : WORD := 4;
	XEXTERNALFAN : BOOL := FALSE;
	XFINISHINSTARTPOS : BOOL := FALSE;
	XUSEAXISPARAMETER : BOOL := FALSE;
END_VAR
VAR_OUTPUT
	XDONE : BOOL;
	XBUSY : BOOL;
	XACTIVE : BOOL;
	XCOMMANDABORTED : BOOL;
	XERROR : BOOL;
	EERRORID : L_IE1P_Error;
	WCYCLESOUT : WORD;
END_VAR
VAR
	FBBRAKESERVICE : POINTER TO L_MC1P_BrakeService;
	FB_BRAKEGRINDIN : L_MC1P_BrakeGrindIn_internal;
	XSTATUS : BOOL;
	DISABLEHOMEPOSCHECK : BOOL;
	GRINDINVELOCITYMODE : BOOL;
END_VAR
END_FUNCTION_BLOCK

(* ---- L_MC1P_BRAKEGRINDIN_INTERNAL.pou ---- *)
FUNCTION_BLOCK L_MC1P_BRAKEGRINDIN_INTERNAL
VAR_INPUT
	XEXECUTE : BOOL;
	EMODE : L_MC1P_GrindInMode := L_MC1P_GrindInMode.CwCcw;
	EADDITIONALLIMITS : L_MC1P_AdditionalLimits := L_MC1P_AdditionalLimits.NotActive;
	LRPOSLIMIT1 : LREAL := 0;
	LRPOSLIMIT2 : LREAL := 0;
	LRMOTORSPEED : LREAL := 60.0;
	LRRAMPTIME : LREAL := 1.0;
	LRONTIME : LREAL := 0.5;
	LROFFTIME : LREAL := 0.5;
	WCYCLES : WORD := 4;
	XCYCLESSETBYPARAMETER : BOOL;
	WCYCLESCW : WORD := 2;
	WCYCLESCCW : WORD := 2;
	XEXTERNALFAN : BOOL := FALSE;
	XFINISHINSTARTPOS : BOOL := FALSE;
	XDISABLEHOMEPOSCHECK : BOOL;
	XGRINDINVELOCITYMODE : BOOL;
END_VAR
VAR_OUTPUT
	XDONE : BOOL;
	XBUSY : BOOL;
	XACTIVE : BOOL;
	XCOMMANDABORTED : BOOL;
	XERROR : BOOL;
	EERRORID : L_IE1P_Error;
	WCYCLESOUT : WORD;
	ESTATE : L_MC1P_BrakeGrindInState := L_MC1P_BrakeGrindInState.NotActive;
END_VAR
VAR
	WFUNID : WORD;
	XEXECUTEOLD : BOOL;
	XRESETOUTPUT : BOOL;
	PAXISREAL : POINTER TO _AXIS_REF_REAL;
	FBBRAKEGI : POINTER TO L_MC1P_BrakeService;
	PBRAKE : POINTER TO L_MC1P_BrakeControl;
	LRGRINDINPOSLOW : LREAL := 0;
	LRGRINDINPOSHIGH : LREAL := 0;
	LRDISTANCE : LREAL := 0;
	LRPOSTOLERANCE : LREAL := 0.1;
	EGRINDINMODEINTERN : L_MC1P_GrindInMode := L_MC1P_GrindInMode.CwCcw;
	READBRAKEPARAMETERS : L_DCO_ReadDriveParameter;
	PDWDUMMY : POINTER TO DWORD;
	PLRDUMMY : POINTER TO LREAL;
	WSTEP : WORD;
	EALLOWEDSERVICEDIRECTION : L_MC1P_ServiceDirection := L_MC1P_ServiceDirection.both;
END_VAR
END_FUNCTION_BLOCK

METHOD CHECKGRINDINDISTANCE
VAR_IN_OUT
	AXIS : AXIS_REF;
	FBBASE : L_MC1P_Template_ForAxis;
END_VAR
END_METHOD

METHOD CHECKVALIDINPUTS
VAR_IN_OUT
	AXIS : AXIS_REF;
	FBBASE : L_MC1P_Template_ForAxis;
END_VAR
END_METHOD

METHOD CHECKVALIDPOSITIONLIMITS
VAR_IN_OUT
	AXIS : AXIS_REF;
	FBBASE : L_MC1P_Template_ForAxis;
END_VAR
END_METHOD

METHOD COPYINPUTSFROMAXISREF
VAR_IN_OUT
	SCPARBRAKEGRINDIN : L_MC1P_BrakeCmdBrakeGrindInPara;
END_VAR
END_METHOD

METHOD MAIN
VAR_IN_OUT
	AXIS : AXIS_REF;
	FBBASE : L_MC1P_Template_ForAxis;
END_VAR
END_METHOD

(* ---- L_MC1P_BRAKEINTERFACE.pou ---- *)
FUNCTION_BLOCK L_MC1P_BRAKEINTERFACE EXTENDS L_MC1P_Template
VAR_INPUT
	XENABLE : BOOL;
	XRELEASEBRAKE : BOOL;
	LRTORQUEADD : LREAL;
	XBRAKEMODEACTIVATE : BOOL;
	EBRAKEMODE : L_MC1P_BrakeMode;
END_VAR
VAR_OUTPUT
	XVALID : BOOL;
	XBUSY : BOOL;
	XERROR : BOOL;
	EERRORID : L_IE1P_Error;
	XBRAKERELEASEOUT : BOOL;
	XBRAKERELEASED : BOOL;
	LRACTTORQUE : LREAL;
	LRSTARTINGTORQUESAVED : LREAL;
	LRSTARTINGTORQUEEFFECTIVE : LREAL;
	EBRAKEMODEACTIVE : L_MC1P_BrakeMode;
END_VAR
VAR
	PAXIS : POINTER TO _AXIS_REF_REAL;
	PBRAKEBASE : POINTER TO L_MC1P_BrakeControlBase;
	PBRAKEADV : POINTER TO L_MC1P_BrakeControl;
	XENABLEOLD : BOOL;
	XSETBRAKEMODEOLD : BOOL;
	EBRAKEMODEOLD : L_MC1P_BrakeMode;
END_VAR
END_FUNCTION_BLOCK

(* ---- L_MC1P_BRAKESERVICE.pou ---- *)
FUNCTION_BLOCK L_MC1P_BRAKESERVICE
VAR_INPUT
	SCPARBRAKEGRINDIN : REFERENCE TO L_MC1P_BrakeCmdBrakeGrindInPara := scParBrakeGrindInit;
	SCPARBRAKETEST : REFERENCE TO L_MC1P_BrakeCmdBrakeTestPara := scParBraketestInit;
END_VAR
VAR_OUTPUT
	XACTIVE : BOOL;
	XDONE : BOOL;
	XERROR : BOOL;
	EERRORID : L_IE1P_Error;
END_VAR
VAR
	SCPARBRAKEGRINDINIT : L_MC1P_BrakeCmdBrakeGrindInPara;
	SCPARBRAKETESTINIT : L_MC1P_BrakeCmdBrakeTestPara;
	ETORQUETESTSEQ : L_MC1P_TorqueTestSequence;
	LRTIMECOUNTER : LREAL;
	LRTIMEVALUE : LREAL;
	WPOWID : WORD;
	XRELEASECINH : BOOL;
	XCINHSTATUS : BOOL;
	XCINHVALID : BOOL;
	WIDENTTORQUESTEP : WORD;
	ECONTROLMODEOLD : L_MC1P_ControlMode;
	LRBTESTTORQUE : LREAL := 0;
	LRBTESTTORQUEMOTOR : LREAL := 0;
	LRBTESTACCTIME : LREAL := 1.0;
	LRBTESTHOLDTIME : LREAL := 4.0;
	LRBTESTPOSFAILTHRESHOLD : LREAL := 0;
	EBTESTDIRECTION : MC_DIRECTION := MC_DIRECTION.mcCurrentDirection;
	EBTESTLOADCOMPENSATIONMODE : L_MC1P_BrakeTestMode := L_MC1P_BrakeTestMode.NoLoadTorque;
	LRBTESTCOMPENSATEDTORQUE : LREAL := 0;
	LRBTESTCOMPENSATEDTORQUEINT : LREAL := 0;
	LRBTESTACTPOSTHRESHOLD : LREAL := 0;
	LRBTESTACTMOTORTORQUE : LREAL := 0;
	EBTESTBRAKETESTSTATE : L_MC1P_BrakeTestState := L_MC1P_BrakeTestState.Init;
	LRFILTERDTORQUE : LREAL;
	LRFILTERCYCLES : LREAL := 5;
	LRFILTERTIMEFACTOR : LREAL;
	DWIDENTCOUNTER : DWORD;
	TORQUETOLERANCE : LREAL := 0.05;
	DWFOLLOWINGERRORZEROCROSSES : DWORD;
	LRACTFOLLOWINGERROROLD : LREAL;
	XCHANGEBRAKEMODETOMANUAL : BOOL;
	XBRAKEINAUTOMODE : BOOL;
	EGRINDINSEQ : L_MC1P_GrindInSequence;
	EGRINDINSEQ_NOEXFAN_NOLIMITS : L_MC1P_GISequence_NoExFan_NoLimits;
	EGRINDINSEQ_NOEXFAN_LIMITS : L_MC1P_GISequence_NoExFan_Limits;
	EGRINDINSEQ_EXFAN_NOLIMITS : L_MC1P_GISequence_ExFan_NoLimits;
	EGRINDINSEQ_EXFAN_LIMITS : L_MC1P_GISequence_ExFan_Limits;
	WGIPULSES : WORD := 10;
	LRTIMECOUNTERMAX : LREAL;
	LRGIVELOCITY : LREAL;
	LRGIRAMPTIME : LREAL;
	LRGIACCELERATION : LREAL;
	LRGITIMEON : LREAL;
	LRGITIMEOFF : LREAL;
	EGIMODE : L_MC1P_GrindInMode;
	EGIADDITIONALLIMITS : L_MC1P_AdditionalLimits;
	LRGIPOSLIMITLOW : LREAL := 0;
	LRGIPOSLIMITHIGH : LREAL := 0;
	XGIEXTERNALFAN : BOOL;
	XGIFINISHINSTARTPOS : BOOL;
	LRMOVEMENTDIRECTION : LREAL := 0;
	XDIRECTIONDETERMINED : BOOL := FALSE;
	L_MC1P_POSPROFILER1 : REFERENCE TO L_Mc1P_PosProfiler;
	SCPROFILEPARAMETER : L_MC1P_ProfileParameter;
	XGIFINISHINSTARTPOSINIT : BOOL := FALSE;
	LRSTARTPOS : LREAL := 0;
	LRGIDISTANCE : LREAL := 0;
	LRGITIMEOFF_TEMP : LREAL := 0;
	LRGITIMEOFF_INIT : LREAL := 0;
	PAXISREAL : POINTER TO _AXIS_REF_REAL;
	WPULSECOUNTERPOS : WORD;
	WPULSECOUNTERNEG : WORD;
	LRGIRAMPTIME_INIT : LREAL;
	LRGIMOVEMENTTIME : LREAL;
	LRGIVELOCITY_TEMP : LREAL;
	LRTIMECOUNTERMAX_INIT : LREAL;
	XPULSESINPOSDIRECTION : BOOL;
	XPULSESINNEGDIRECTION : BOOL;
	XSTARTLIMITSWITCHTIMECOUNTER : BOOL;
	LRLIMITSWITCHTIMECOUNTER : LREAL;
	LRTIMECOUNTERMAX_TEMP : LREAL;
	LRGIMOVEMENTTIME_TEMP : LREAL;
	WCYCLESOUT : WORD;
	STTORQUETESTMONITORING : L_MC1P_TorqueTestMonitoring;
	LRTORQUETESTPT1DELAY : LREAL := 0.01;
	LRTORQUETOLERANCEPCT : LREAL := 0.1;
	LRSETTORQUETMP : LREAL;
	LRDIFF : LREAL;
	XPOSPROFILERINUSE : BOOL;
	LRMEANVALUE : LREAL;
	LRVALUECOUNTER : LREAL;
	LRVARIANCE : LREAL;
	LRSTD : LREAL;
	LRSTDOLD : LREAL;
	LRDIFF2 : LREAL;
	_XGRINDINVELOCITYMODE : BOOL;
	POSPROFILERINUSE : BOOL;
	TORQUETEST_BRAKEINAUTOMODE : BOOL;
	TORQUETEST_CHANGEBRAKEMODETOMANUAL : BOOL;
END_VAR
END_FUNCTION_BLOCK

METHOD CHECKDISTANCE_EXFAN_LIMITS
VAR_IN_OUT
	AXIS : Axis_Ref;
	BRAKE : L_MC1P_BrakeControl;
END_VAR
END_METHOD

METHOD CHECKDISTANCE_NOEXFAN_LIMITS
VAR_IN_OUT
	AXIS : Axis_Ref;
	BRAKE : L_MC1P_BrakeControl;
END_VAR
END_METHOD

METHOD GI_GENERATERAMP : BOOL
VAR_INPUT
	LRENDVELOCITY : LREAL := 0;
END_VAR
VAR_IN_OUT
	AXIS : _AXIS_REF_REAL;
END_VAR
END_METHOD

METHOD GENERATEPULSE : BOOL
VAR_IN_OUT
	AXIS : _AXIS_REF_REAL;
	BRAKE : L_MC1P_BrakeControl;
END_VAR
END_METHOD

METHOD GRINDIN_EXIT
VAR_IN_OUT
	BRAKE : L_MC1P_BrakeControl;
	AXIS : _AXIS_REF_REAL;
END_VAR
END_METHOD

METHOD GRINDIN_INIT
END_METHOD

METHOD GRINDIN_MAIN
VAR_IN_OUT
	BRAKE : L_MC1P_BrakeControl;
	AXIS : _AXIS_REF_REAL;
END_VAR
END_METHOD

METHOD GRINDIN_SETPARAMETER
VAR_INPUT
	LRSPEED : LREAL := 0;
	LRRAMPTIME : LREAL := 0;
	EMODE : L_MC1P_GrindInMode := 0;
	EADDITIONALLIMITS : L_MC1P_AdditionalLimits := L_MC1P_AdditionalLimits.NotActive;
	LRTIMEON : LREAL := 1.0;
	LRTIMEOFF : LREAL := 4.0;
	WCYCLES : WORD := 4;
	WCYCLESCW : WORD := 4;
	WCYCLESCCW : WORD := 4;
	LRGRINDINPOSLIMIT1 : LREAL := 0;
	LRGRINDINPOSLIMIT2 : LREAL := 0;
	XEXTERNALFAN : BOOL;
	XFINISHINSTARTPOS : BOOL;
	XCYCLESSETBYPARAMETER : BOOL := FALSE;
	XGRINDINVELOCITYMODE : BOOL;
END_VAR
VAR_IN_OUT
	AXIS : _AXIS_REF_REAL;
END_VAR
END_METHOD

METHOD SETPULSES
VAR_INPUT
	XCYCLESSETBYPARAMETER : BOOL;
	WCYCLES : WORD;
	WCYCLESCW : WORD;
	WCYCLESCCW : WORD;
END_VAR
END_METHOD

METHOD STEPSEQUENCE1_NOEXFAN_NOLIMITS
VAR_INPUT
	BRAKESWITCH : L_MC1P_BrakeState;
END_VAR
VAR_IN_OUT
	BRAKE : L_MC1P_BrakeControl;
	AXIS : _AXIS_REF_REAL;
END_VAR
END_METHOD

METHOD STEPSEQUENCE2_NOEXFAN_LIMITS
VAR_INPUT
	BRAKESWITCH : L_MC1P_BrakeState;
END_VAR
VAR_IN_OUT
	BRAKE : L_MC1P_BrakeControl;
	AXIS : _AXIS_REF_REAL;
END_VAR
END_METHOD

METHOD STEPSEQUENCE3_EXFAN_NOLIMITS
VAR_INPUT
	BRAKESWITCH : L_MC1P_BrakeState;
END_VAR
VAR_IN_OUT
	BRAKE : L_MC1P_BrakeControl;
	AXIS : _AXIS_REF_REAL;
END_VAR
END_METHOD

METHOD STEPSEQUENCE4_EXFAN_LIMITS
VAR_INPUT
	BRAKESWITCH : L_MC1P_BrakeState;
END_VAR
VAR_IN_OUT
	BRAKE : L_MC1P_BrakeControl;
	AXIS : _AXIS_REF_REAL;
END_VAR
END_METHOD

METHOD CALCSTATISTICVALUES
VAR_INPUT
	LRNEWVALUE : LREAL;
END_VAR
VAR_IN_OUT
	LRMEANVALUE : LREAL;
	LRVALUECOUNTER : LREAL;
	LRVARIANCE : LREAL;
	LRSTD : LREAL;
END_VAR
END_METHOD

METHOD TORQUETEST_EXIT
VAR_IN_OUT
	BRAKE : L_MC1P_BrakeControlBase;
	AXIS : _AXIS_REF_REAL;
END_VAR
END_METHOD

METHOD TORQUETEST_IDENTTORQUE : BOOL
VAR_INPUT
	BRAKESWITCH : L_MC1P_BrakeState;
END_VAR
VAR_IN_OUT
	BRAKE : L_MC1P_BrakeControlBase;
	AXIS : _AXIS_REF_REAL;
END_VAR
END_METHOD

METHOD TORQUETEST_INIT
END_METHOD

METHOD TORQUETEST_MAIN
VAR_IN_OUT
	BRAKE : L_MC1P_BrakeControlBase;
	AXIS : _AXIS_REF_REAL;
END_VAR
END_METHOD

METHOD TORQUETEST_MONITORING : BOOL
VAR_INPUT
	LRPT1DELAY : LREAL;
	LRTORQUETOLERANCE : LREAL;
END_VAR
VAR_IN_OUT
	AXIS : _AXIS_REF_REAL;
END_VAR
END_METHOD

METHOD TORQUETEST_SETPARAMETER
VAR_INPUT
	LRTORQUE : LREAL := 0;
	LRACCTIME : LREAL := 1.0;
	LRHOLDTIME : LREAL := 4.0;
	LRPOSFAILTHRESHOLD : LREAL := 0;
	EDIRECTION : MC_DIRECTION := MC_DIRECTION.mcCurrentDirection;
	ELOADCOMPENSATIONMODE : L_MC1P_BrakeTestMode := L_MC1P_BrakeTestMode.NoLoadTorque;
END_VAR
END_METHOD

(* ---- L_MC1P_BRAKETEST.pou ---- *)
FUNCTION_BLOCK L_MC1P_BRAKETEST EXTENDS L_MC1P_Template
VAR_INPUT
	XEXECUTE : BOOL;
	LRMOTORTORQUE : LREAL := 0;
	LRRAMPTIME : LREAL := 1.0;
	LRHOLDTIME : LREAL := 4.0;
	LRPOSTHRESHOLD : LREAL;
	EDIRECTION : MC_DIRECTION := MC_DIRECTION.mcCurrentDirection;
	EMODE : L_MC1P_BrakeTestMode := L_MC1P_BrakeTestMode.NoLoadTorque;
	XUSEAXISPARAMETER : BOOL := FALSE;
END_VAR
VAR_OUTPUT
	XDONE : BOOL;
	XBUSY : BOOL;
	XACTIVE : BOOL;
	XCOMMANDABORTED : BOOL;
	XERROR : BOOL;
	EERRORID : L_IE1P_Error;
	LRIDENTIFIEDTORQUE : LREAL;
	LRACTPOSTHRESHOLD : LREAL;
	LRACTMOTORTORQUE : LREAL;
	ESTATE : L_MC1P_BrakeTestState := L_MC1P_BrakeTestState.NotActive;
END_VAR
VAR
	FBBRAKESERVICE : POINTER TO L_MC1P_BrakeService;
	FB_BRAKETEST : L_MC1P_BrakeTest_internal;
	XSTATUS : BOOL;
END_VAR
END_FUNCTION_BLOCK

(* ---- L_MC1P_BRAKETEST_INTERNAL.pou ---- *)
FUNCTION_BLOCK L_MC1P_BRAKETEST_INTERNAL
VAR_INPUT
	XEXECUTE : BOOL;
	LRMOTORTORQUE : LREAL := 0;
	LRRAMPTIME : LREAL := 1.0;
	LRHOLDTIME : LREAL := 4.0;
	LRPOSTHRESHOLD : LREAL;
	EDIRECTION : MC_DIRECTION := MC_DIRECTION.mcCurrentDirection;
	EMODE : L_MC1P_BrakeTestMode := L_MC1P_BrakeTestMode.NoLoadTorque;
END_VAR
VAR_OUTPUT
	XDONE : BOOL;
	XBUSY : BOOL;
	XACTIVE : BOOL;
	XCOMMANDABORTED : BOOL;
	XERROR : BOOL;
	EERRORID : L_IE1P_Error;
	LRIDENTIFIEDTORQUE : LREAL;
	LRACTPOSTHRESHOLD : LREAL;
	LRACTMOTORTORQUE : LREAL;
	ESTATE : L_MC1P_BrakeTestState := L_MC1P_BrakeTestState.NotActive;
END_VAR
VAR
	WFUNID : WORD;
	XEXECUTEOLD : BOOL;
	XRESETOUTPUT : BOOL;
	PAXISREAL : POINTER TO _AXIS_REF_REAL;
	FBBRAKETEST : POINTER TO L_MC1P_BrakeService;
	PBRAKE : POINTER TO L_MC1P_BrakeControlBase;
	WSTEP : WORD;
	READBRAKEPARAMETERS : L_DCO_ReadDriveParameter;
	PDWDUMMY : POINTER TO DWORD;
	XBRAKELOGICINDRIVE : BOOL;
	XBRAKEINAUTOMODE : BOOL;
END_VAR
END_FUNCTION_BLOCK

METHOD COPYINPUTSFROMAXISREF
VAR_IN_OUT
	SCPARBRAKETEST : L_MC1P_BrakeCmdBrakeTestPara;
END_VAR
END_METHOD

METHOD MAIN
VAR_IN_OUT
	AXIS : AXIS_REF;
	FBBASE : L_MC1P_Template_ForAxis;
END_VAR
END_METHOD

(* ---- L_MC1P_BUTTERWORTHENCODERPOSFILTER.pou ---- *)
FUNCTION_BLOCK L_MC1P_BUTTERWORTHENCODERPOSFILTER
VAR_INPUT
	LRFILTERTIME : LREAL;
	XCALCULATEVEL : BOOL;
END_VAR
VAR
	FB_BUTTERWORTHFILTER : L_USPP_Butterworth2ndOrder;
	LRTASKCYCLEINT : LREAL;
	LRTASKCYCLEINV : LREAL;
	LRFILTERTIMEOLD : LREAL;
	LRCYCPOSINSTORED : LREAL;
	LRCYCPOSOUTOLD : LREAL;
	LRCYCPOSINOLD : LREAL;
	LRROUNDS : LREAL;
END_VAR
END_FUNCTION_BLOCK

METHOD CALCULATE
VAR_INPUT
	LRCYCPOSIN : LREAL;
	LRCYCVELIN : LREAL;
END_VAR
VAR_OUTPUT
	LRCYCPOSOUT : LREAL;
	LRCYCVELOUT : LREAL;
	WFILTERSTATE : WORD;
END_VAR
END_METHOD

METHOD DETECTOVERFLOW
VAR_INPUT
	LRACTPOS : LREAL;
	LRPOSOLD : LREAL;
	LRCYCLELENGTH : LREAL;
END_VAR
VAR_IN_OUT
	LRACTCOUNTER : LREAL;
END_VAR
END_METHOD

METHOD INIT
END_METHOD

METHOD RESETINTERNAL
END_METHOD

METHOD RESET
END_METHOD

METHOD FB_INIT : BOOL
VAR_INPUT
	BINITRETAINS : BOOL;
	BINCOPYCODE : BOOL;
END_VAR
END_METHOD

(* ---- L_MC1P_CHANGEABLE.pou ---- *)
FUNCTION_BLOCK L_MC1P_CHANGEABLE
VAR
	DWID : DWORD := 0;
	ID : DWORD;
END_VAR
END_FUNCTION_BLOCK

METHOD ASSIGNID
VAR_INPUT
	DWID : DWORD;
END_VAR
END_METHOD

METHOD CHANGE : BOOL
END_METHOD

METHOD CHANGED : BOOL
VAR_INPUT
	DWID : DWORD;
END_VAR
END_METHOD

METHOD INITID
END_METHOD

(* ---- L_MC1P_CHANGEMACHINEDATA.pou ---- *)
FUNCTION_BLOCK L_MC1P_CHANGEMACHINEDATA EXTENDS L_MC1P_Template
VAR_INPUT
	XEXECUTE : BOOL;
	XSETFEEDCONSTANT : BOOL;
	LRFEEDCONSTANT : LREAL := 360.0;
	XSETGEARFACTOR : BOOL;
	DWGEARDENOMINATOR : DWORD := 1;
	DWGEARNUMERATOR : DWORD := 1;
	XSETADDGEARFACTOR : BOOL;
	DWADDGEARDENOMINATOR : DWORD := 1;
	DWADDGEARNUMERATOR : DWORD := 1;
	XSETPOSRESOLUTION : BOOL;
	DWPOSRESOLUTION : DWORD := 65536;
	XSETORIENTATION : BOOL;
	XORIENTATION : BOOL := FALSE;
	XSETTRAVERSINGRANGE : BOOL;
	ETRAVERSINGRANGE : L_MC1P_TraversingRange := L_MC1P_TraversingRange.Limited;
	XSETCYCLELENGTH : BOOL;
	LRCYCLELENGTH : LREAL := 360.0;
END_VAR
VAR_OUTPUT
	XDONE : BOOL;
	XBUSY : BOOL;
	XERROR : BOOL;
	EERRORID : L_IE1P_Error;
END_VAR
VAR
	XEXECUTEOLD : BOOL;
	LRFEEDCONSTANTNEW : LREAL := 360.0;
	DWGEARDENOMINATORNEW : DWORD := 1;
	DWGEARNUMERATORNEW : DWORD := 1;
	DWADDGEARDENOMINATORNEW : DWORD := 1;
	DWADDGEARNUMERATORNEW : DWORD := 1;
	DWPOSRESOLUTIONNEW : DWORD := 65536;
	XORIENTATIONNEW : BOOL := FALSE;
	ETRAVERSINGRANGENEW : L_MC1P_TraversingRange := L_MC1P_TraversingRange.Limited;
	LRCYCLELENGTHNEW : LREAL := 360.0;
	XCHANGES : BOOL;
	XREINIT : BOOL;
	PAXISREAL : POINTER TO _AXIS_REF_REAL;
	PWDUMMY1 : POINTER TO WORD;
	PWDUMMY2 : POINTER TO WORD;
	PXDUMMY : POINTER TO BOOL;
	XWRITEPOSRESOLUTION : BOOL;
	ITIMEOUTCNT : INT;
	PBRAKE : POINTER TO L_MC1P_BrakeControlBase;
END_VAR
END_FUNCTION_BLOCK

METHOD SETTIMEOUTCNT
VAR_IN_OUT
	AXIS : AXIS_REF;
END_VAR
END_METHOD

(* ---- L_MC1P_CINHHANDLING.pou ---- *)
FUNCTION_BLOCK L_MC1P_CINHHANDLING EXTENDS L_MC1P_Template
VAR_INPUT
	XENABLE : BOOL;
	XSTAYINLASTSTATE : BOOL;
	XMOVELASTSETPOS : BOOL;
	LRWINDOWPOS : LREAL;
	LRWINDOWNEG : LREAL;
	LRSETVEL : LREAL;
	LRSETACC : LREAL;
	LRSETDEC : LREAL;
	LRSETJERK : LREAL;
	EDIRECTION : MC_DIRECTION;
END_VAR
VAR_OUTPUT
	XDONE : BOOL;
	XBUSY : BOOL;
	XACTIVE : BOOL;
	XERROR : BOOL;
	EERRORID : L_IE1P_Error;
	XREADYTOCONTINUE : BOOL;
	XINSIDEPOSWINDOW : BOOL;
	XINSIDEACTPOSWINDOW : BOOL;
	EAXISSTATEREAL : L_MC1P_AXIS_STATE := L_MC1P_AXIS_STATE.Disabled;
	LRDISTANCE : LREAL;
END_VAR
VAR
	XENABLEOLD : BOOL;
	PXDUMMY : POINTER TO BOOL;
END_VAR
END_FUNCTION_BLOCK

(* ---- L_MC1P_CLUTCHVELOCITY.pou ---- *)
FUNCTION_BLOCK L_MC1P_CLUTCHVELOCITY
VAR_INPUT
	XENABLE : BOOL;
	XCLOSE : BOOL;
	XOPENINSTANT : BOOL;
	LRCYCVEL : LREAL;
	LRGROUNDVEL : LREAL;
	LRACCDECOPEN : LREAL;
	LRACCDECCLOSE : LREAL;
	LRDECSTOP : LREAL;
	LRJERK : LREAL;
END_VAR
VAR_OUTPUT
	XOPEN : BOOL;
	XACCDEC : BOOL;
	LRSETVELOUT : LREAL;
END_VAR
VAR
	HLP_CLUTCHV : L_MC1P_HlpRampGenerator;
	LRBASESPEED : LREAL;
	LRCLOSESPEED : LREAL;
	LRNUMERATOR : LREAL;
	LRDENUMERATOR : LREAL;
	XINITFLAG : BOOL;
	DNSTATE : DINT;
	WSTEPCOUNTER : WORD;
	LRSETVELRAMPGENERATOR : LREAL;
	LRLOADRAMPGENDIFF : LREAL;
	CLUTCHV_INIT : WORD := 0;
	CLUTCHV_ENABLE : WORD := 1;
	CLUTCHV_CLOSE : WORD := 2;
	CLUTCHV_CLOSING : WORD := 3;
	CLUTCHV_CLOSE_DONE : WORD := 4;
	CLUTCHV_OPENING : WORD := 5;
	CLUTCHV_OPEN_STOP : WORD := 6;
	CLUTCHV_OPENINSTANT_DONE : WORD := 7;
	CLUTCHV_OPENINSTANT_DISABLE : WORD := 8;
	CLUTCHV_CLOSING_STOP : WORD := 9;
END_VAR
END_FUNCTION_BLOCK

METHOD CLUTCHCLOSINGTRANSITION
END_METHOD

METHOD CLUTCHOPENINGTRANSITION
END_METHOD

METHOD OPENINSTANTTRANSITION
END_METHOD

(* ---- L_MC1P_COMMCAN.pou ---- *)
FUNCTION_BLOCK L_MC1P_COMMCAN
VAR
	AFBPARREAD : ARRAY [1..c_SdoMaxNum] OF CiA405.SDO_READ;
	AFBPARWRITE : ARRAY [1..c_SdoMaxNum] OF CiA405.SDO_WRITE;
	FBCOMMSTATE : CiA405.GET_STATE;
	FBCOMMNMT : CiA405.NMT;
	SZSIZEREAD : UINT;
	ECOMMSTATE_INT : L_DCO.L_DCO_CommState;
	C_SDOMAXNUM : WORD := 10;
	COMPONENTINFOSUPPORTED : BOOL;
	SIMULATIONINTERFACE : L_MC1P_ICommmunicationSimulation;
	SLAVEDEVICEMODULEHANDLER : L_IMHP_IModuleHandler;
END_VAR
END_FUNCTION_BLOCK

METHOD FORWARDERROR
VAR_INPUT
	XENABLE : BOOL;
	XWARNING : BOOL;
	XERROR : BOOL;
	WERRORID : WORD;
	WTEXTREFID : WORD;
	XRESETERROR : BOOL := FALSE;
	AXISMODULEHANDLER : L_IMHP_IModuleHandler;
END_VAR
END_METHOD

METHOD GETCOMMPARAMETER
VAR_INPUT
	PCONNECTOR : POINTER TO IoStandard.IoConfigConnector;
END_VAR
VAR_OUTPUT
	PSLAVECONNECTOR : POINTER TO IoStandard.IoConfigConnector;
	UINETID : UINT;
	UIDEVICEID : UINT;
	XSENDFRAMEATTASKSTART : BOOL;
	UDIPRODUCTCODE : DWORD;
	PMASTERCONNECTOR : POINTER TO IoStandard.IoConfigConnector;
END_VAR
END_METHOD

METHOD GETCOMMSTATE : L_DCO.L_DCO_CommState
VAR_INPUT
	PAXISCOMM : POINTER TO _AXIS_REF_COM;
END_VAR
END_METHOD

METHOD GETPDINEQPDOUT : BOOL
END_METHOD

METHOD GETSDOERROR : WORD
VAR_INPUT
	DWERRORCODE : DWORD;
	DWERRORINFO : DWORD;
END_VAR
END_METHOD

METHOD PARREAD
VAR_INPUT
	WIDX : DWORD;
END_VAR
END_METHOD

METHOD PARREAD_GETOUTPUT
VAR_INPUT
	WIDX : DWORD;
END_VAR
VAR_OUTPUT
	SZDATAREAD : CAA_SIZE;
	XDONE : BOOL;
	XERROR : BOOL;
	WERROR : WORD;
END_VAR
END_METHOD

METHOD PARREAD_SETINPUT
VAR_INPUT
	WIDX : DWORD;
	XEXECUTE : BOOL;
	WINDEX : WORD;
	BYSUBINDEX : BYTE;
	PBUFFER : POINTER TO BYTE;
	SZSIZE : UDINT;
	UDITIMEOUT : UDINT;
END_VAR
END_METHOD

METHOD PARWRITE
VAR_INPUT
	WIDX : DWORD;
END_VAR
END_METHOD

METHOD PARWRITE_GETOUTPUT
VAR_INPUT
	WIDX : DWORD;
END_VAR
VAR_OUTPUT
	XDONE : BOOL;
	XERROR : BOOL;
	WERROR : WORD;
END_VAR
END_METHOD

METHOD PARWRITE_SETINPUT
VAR_INPUT
	WIDX : DWORD;
	XEXECUTE : BOOL;
	WINDEX : WORD;
	BYSUBINDEX : BYTE;
	PBUFFER : POINTER TO BYTE;
	SZSIZE : UDINT;
	UDITIMEOUT : UDINT;
END_VAR
END_METHOD

METHOD RESET
END_METHOD

METHOD RESTARTMASTER
VAR_INPUT
	XEXECUTE : BOOL;
	PAXIS : POINTER TO _AXIS_REF_COM;
END_VAR
VAR_OUTPUT
	XDONE : BOOL;
	XERROR : BOOL;
	XBUSY : BOOL;
	DWERROR : DWORD;
END_VAR
END_METHOD

METHOD SETBASICINITIALISATION
VAR_IN_OUT
	AXIS : _AXIS_REF_REAL;
END_VAR
END_METHOD

METHOD SETCOMPONENTINFO
VAR_INPUT
	DATASELECTION : WORD;
	SDATA : STRING;
END_VAR
END_METHOD

(* ---- L_MC1P_COMMECAT.pou ---- *)
FUNCTION_BLOCK L_MC1P_COMMECAT
VAR_INPUT
	XSLOTB : BOOL := FALSE;
	ITFSLAVEMULTIAXISMODULEHANDLER : L_IMHP_IModuleHandler;
END_VAR
VAR
	WCONNECTORTYPE : WORD;
	XFIRSTSLAVEDETECTION : BOOL := TRUE;
	AFBPARREAD : ARRAY [1..c_SdoMaxNum] OF L_ETC_CoE_SdoRead;
	AFBPARWRITE : ARRAY [1..c_SdoMaxNum] OF L_ETC_CoE_SdoWrite;
	SLAVE : POINTER TO ETCSlave;
	SLAVEMODULEHANDLER : L_IMHP_IModuleHandler;
	FBRESTARTMASTER : L_MC1P_ResetMaster_ETC;
	PPDIN : POINTER TO BYTE;
	PPDOUT : POINTER TO BYTE;
	PWOUTPUTDATAOLD : ARRAY [0..1] OF WORD;
	L_IE1P_FORWARDERROR1 : L_IE1P_ForwardError;
	XCOMPONENTINFOSUPPORTED : BOOL := FALSE;
	M_UINETID : UINT;
	M_UIDEVICEID : UINT;
	ITFCOMMSIMULATION : L_MC1P_ICommmunicationSimulation;
	XUSEFIRSTAXISFORCOMMCHECK : BOOL;
	C_SDOMAXNUM : WORD := 10;
	COMPONENTINFOSUPPORTED : BOOL;
	SIMULATIONINTERFACE : L_MC1P_ICommmunicationSimulation;
	SLAVEDEVICEMODULEHANDLER : L_IMHP_IModuleHandler;
END_VAR
END_FUNCTION_BLOCK

METHOD CONVERTSTATE : WORD
VAR_INPUT
	WSTATE : WORD;
END_VAR
END_METHOD

METHOD FINDMASTERCONNECTOR : POINTER TO IoStandard.IoConfigConnector
VAR_INPUT
	PSLAVECONNECTOR : POINTER TO IoStandard.IoConfigConnector;
END_VAR
END_METHOD

METHOD FORWARDERROR
VAR_INPUT
	XENABLE : BOOL;
	XWARNING : BOOL;
	XERROR : BOOL;
	WERRORID : WORD;
	WTEXTREFID : WORD;
	XRESETERROR : BOOL := FALSE;
	AXISMODULEHANDLER : L_IMHP_IModuleHandler;
END_VAR
END_METHOD

METHOD GETADRESSFORCOMMCHECK
VAR_INPUT
	PCONNECTOR : POINTER TO IoConfigConnector;
END_VAR
END_METHOD

METHOD GETCOMMPARAMETER
VAR_INPUT
	PCONNECTOR : POINTER TO IoStandard.IoConfigConnector;
END_VAR
VAR_OUTPUT
	PSLAVECONNECTOR : POINTER TO IoStandard.IoConfigConnector;
	UINETID : UINT;
	UIDEVICEID : UINT;
	XSENDFRAMEATTASKSTART : BOOL;
	UDIPRODUCTCODE : DWORD;
	PMASTERCONNECTOR : POINTER TO IoStandard.IoConfigConnector;
END_VAR
END_METHOD

METHOD GETCOMMSTATE : L_DCO.L_DCO_CommState
VAR_INPUT
	PAXISCOMM : POINTER TO _AXIS_REF_COM;
END_VAR
END_METHOD

METHOD GETPDINEQPDOUT : BOOL
END_METHOD

METHOD GETSDOERROR : WORD
VAR_INPUT
	DWERRORCODE : DWORD;
END_VAR
END_METHOD

METHOD PARREAD
VAR_INPUT
	WIDX : DWORD;
END_VAR
END_METHOD

METHOD PARREAD_GETOUTPUT
VAR_INPUT
	WIDX : DWORD;
END_VAR
VAR_OUTPUT
	SZDATAREAD : CAA_SIZE;
	XDONE : BOOL;
	XERROR : BOOL;
	WERROR : WORD;
END_VAR
END_METHOD

METHOD PARREAD_SETINPUT
VAR_INPUT
	WIDX : DWORD;
	XEXECUTE : BOOL;
	WINDEX : WORD;
	BYSUBINDEX : BYTE;
	PBUFFER : POINTER TO BYTE;
	SZSIZE : UDINT;
	UDITIMEOUT : UDINT;
END_VAR
END_METHOD

METHOD PARWRITE
VAR_INPUT
	WIDX : DWORD;
END_VAR
END_METHOD

METHOD PARWRITE_GETOUTPUT
VAR_INPUT
	WIDX : DWORD;
END_VAR
VAR_OUTPUT
	XDONE : BOOL;
	XERROR : BOOL;
	WERROR : WORD;
END_VAR
END_METHOD

METHOD PARWRITE_SETINPUT
VAR_INPUT
	WIDX : DWORD;
	XEXECUTE : BOOL;
	WINDEX : WORD;
	BYSUBINDEX : BYTE;
	PBUFFER : POINTER TO BYTE;
	SZSIZE : UDINT;
	UDITIMEOUT : UDINT;
END_VAR
END_METHOD

METHOD RESET
END_METHOD

METHOD RESTARTMASTER
VAR_INPUT
	XEXECUTE : BOOL;
	PAXIS : POINTER TO _AXIS_REF_COM;
END_VAR
VAR_OUTPUT
	XDONE : BOOL;
	XERROR : BOOL;
	XBUSY : BOOL;
	DWERROR : DWORD;
END_VAR
END_METHOD

METHOD SETBASICINITIALISATION
VAR_IN_OUT
	AXIS : _AXIS_REF_REAL;
END_VAR
END_METHOD

METHOD SETCOMPONENTINFO
VAR_INPUT
	DATASELECTION : WORD;
	SDATA : STRING;
END_VAR
END_METHOD

(* ---- L_MC1P_COMMI900.pou ---- *)
FUNCTION_BLOCK L_MC1P_COMMI900
VAR_INPUT
	XDIRECTREADACCESSTOBASEFIRMWARE : BOOL := FALSE;
	XDIRECTWRITEACCESSTOBASEFIRMWARE : BOOL := FALSE;
END_VAR
VAR
	AFBPARREAD : ARRAY [1..c_SdoMaxNum] OF L_IPAP_ParameterRead;
	AFBPARWRITE : ARRAY [1..c_SdoMaxNum] OF L_IPAP_ParameterWrite;
	XRESTARTOLD : BOOL;
	ITFCOMMSIMULATION : L_MC1P_ICommmunicationSimulation;
	C_SDOMAXNUM : WORD := 10;
	COMPONENTINFOSUPPORTED : BOOL;
	SIMULATIONINTERFACE : L_MC1P_ICommmunicationSimulation;
	SLAVEDEVICEMODULEHANDLER : L_IMHP_IModuleHandler;
END_VAR
END_FUNCTION_BLOCK

METHOD CONVERTSTATE : WORD
VAR_INPUT
	WSTATE : WORD;
END_VAR
END_METHOD

METHOD FORWARDERROR
VAR_INPUT
	XENABLE : BOOL;
	XWARNING : BOOL;
	XERROR : BOOL;
	WERRORID : WORD;
	WTEXTREFID : WORD;
	XRESETERROR : BOOL := FALSE;
	AXISMODULEHANDLER : L_IMHP_IModuleHandler;
END_VAR
END_METHOD

METHOD GETCOMMPARAMETER
VAR_INPUT
	PCONNECTOR : POINTER TO IoStandard.IoConfigConnector;
END_VAR
VAR_OUTPUT
	PSLAVECONNECTOR : POINTER TO IoStandard.IoConfigConnector;
	UINETID : UINT;
	UIDEVICEID : UINT;
	XSENDFRAMEATTASKSTART : BOOL;
	UDIPRODUCTCODE : DWORD;
	PMASTERCONNECTOR : POINTER TO IoStandard.IoConfigConnector;
END_VAR
END_METHOD

METHOD GETCOMMSTATE : L_DCO.L_DCO_CommState
VAR_INPUT
	PAXISCOMM : POINTER TO _AXIS_REF_COM;
END_VAR
END_METHOD

METHOD GETPDINEQPDOUT : BOOL
END_METHOD

METHOD GETSDOERROR : WORD
VAR_INPUT
	DWERRORCODE : DWORD;
END_VAR
END_METHOD

METHOD PARREAD
VAR_INPUT
	WIDX : DWORD;
END_VAR
END_METHOD

METHOD PARREAD_GETOUTPUT
VAR_INPUT
	WIDX : DWORD;
END_VAR
VAR_OUTPUT
	SZDATAREAD : CAA_SIZE;
	XDONE : BOOL;
	XERROR : BOOL;
	WERROR : WORD;
END_VAR
END_METHOD

METHOD PARREAD_SETINPUT
VAR_INPUT
	WIDX : DWORD;
	XEXECUTE : BOOL;
	WINDEX : WORD;
	BYSUBINDEX : BYTE;
	PBUFFER : POINTER TO BYTE;
	SZSIZE : UDINT;
	UDITIMEOUT : UDINT;
END_VAR
END_METHOD

METHOD PARWRITE
VAR_INPUT
	WIDX : DWORD;
END_VAR
END_METHOD

METHOD PARWRITE_GETOUTPUT
VAR_INPUT
	WIDX : DWORD;
END_VAR
VAR_OUTPUT
	XDONE : BOOL;
	XERROR : BOOL;
	WERROR : WORD;
END_VAR
END_METHOD

METHOD PARWRITE_SETINPUT
VAR_INPUT
	WIDX : DWORD;
	XEXECUTE : BOOL;
	WINDEX : WORD;
	BYSUBINDEX : BYTE;
	PBUFFER : POINTER TO BYTE;
	SZSIZE : UDINT;
	UDITIMEOUT : UDINT;
END_VAR
END_METHOD

METHOD RESET
END_METHOD

METHOD RESTARTMASTER
VAR_INPUT
	XEXECUTE : BOOL;
	PAXIS : POINTER TO _AXIS_REF_COM;
END_VAR
VAR_OUTPUT
	XDONE : BOOL;
	XERROR : BOOL;
	XBUSY : BOOL;
	DWERROR : DWORD;
END_VAR
END_METHOD

METHOD SETBASICINITIALISATION
VAR_IN_OUT
	AXIS : _AXIS_REF_REAL;
END_VAR
END_METHOD

METHOD SETCOMPONENTINFO
VAR_INPUT
	DATASELECTION : WORD;
	SDATA : STRING;
END_VAR
END_METHOD

(* ---- L_MC1P_COMMSIM.pou ---- *)
FUNCTION_BLOCK L_MC1P_COMMSIM
VAR_INPUT
	LRTASKCYCLE : LREAL;
	XOPERATIONAL : BOOL;
	WPARAMDATACOUNT : WORD;
	PPARAMDATA : POINTER TO L_MC1P_ParameterDataSim;
END_VAR
VAR
	AFBPARREAD : ARRAY [1..c_SdoMaxNum] OF L_MC1P_ParSimRead;
	AFBPARWRITE : ARRAY [1..c_SdoMaxNum] OF L_MC1P_ParSimWrite;
	XRESTARTOLD : BOOL;
	ERRORREAD : L_MC1P_ParameterDataSim;
	ERRORWRITE : L_MC1P_ParameterDataSim;
	C_SDOMAXNUM : WORD := 10;
END_VAR
END_FUNCTION_BLOCK

METHOD GETCOMMSTATE : L_DCO.L_DCO_CommState
VAR_INPUT
	PAXISCOMM : POINTER TO _AXIS_REF_COM;
END_VAR
END_METHOD

METHOD GETSDOERROR : WORD
VAR_INPUT
	DWERRORCODE : DWORD;
END_VAR
END_METHOD

METHOD PARREAD
VAR_INPUT
	WIDX : DWORD;
END_VAR
END_METHOD

METHOD PARREAD_GETOUTPUT
VAR_INPUT
	WIDX : DWORD;
END_VAR
VAR_OUTPUT
	SZDATAREAD : CAA_SIZE;
	XDONE : BOOL;
	XERROR : BOOL;
	WERROR : WORD;
END_VAR
END_METHOD

METHOD PARREAD_SETINPUT
VAR_INPUT
	WIDX : DWORD;
	XEXECUTE : BOOL;
	WINDEX : WORD;
	BYSUBINDEX : BYTE;
	PBUFFER : POINTER TO BYTE;
	SZSIZE : UDINT;
	UDITIMEOUT : UDINT;
	XSLOTB : BOOL;
END_VAR
END_METHOD

METHOD PARWRITE
VAR_INPUT
	WIDX : DWORD;
END_VAR
END_METHOD

METHOD PARWRITE_GETOUTPUT
VAR_INPUT
	WIDX : DWORD;
END_VAR
VAR_OUTPUT
	XDONE : BOOL;
	XERROR : BOOL;
	WERROR : WORD;
END_VAR
END_METHOD

METHOD PARWRITE_SETINPUT
VAR_INPUT
	WIDX : DWORD;
	XEXECUTE : BOOL;
	WINDEX : WORD;
	BYSUBINDEX : BYTE;
	PBUFFER : POINTER TO BYTE;
	SZSIZE : UDINT;
	UDITIMEOUT : UDINT;
	XSLOTB : BOOL;
END_VAR
END_METHOD

METHOD RESTARTMASTER
VAR_INPUT
	XEXECUTE : BOOL;
	PAXIS : POINTER TO _AXIS_REF_COM;
END_VAR
VAR_OUTPUT
	XDONE : BOOL;
	XERROR : BOOL;
	XBUSY : BOOL;
	DWERROR : DWORD;
END_VAR
END_METHOD

(* ---- L_MC1P_COMPENSATIONBASE.pou ---- *)
FUNCTION_BLOCK L_MC1P_COMPENSATIONBASE EXTENDS L_MC1P_ManipulationBase
END_FUNCTION_BLOCK

METHOD CONNECTTOAXIS
VAR_IN_OUT
	AXIS : Axis_Ref;
END_VAR
END_METHOD

METHOD DISCONNECTFROMAXIS
VAR_IN_OUT
	AXIS : Axis_Ref;
END_VAR
END_METHOD

METHOD FILTERSTARTCONDITION
VAR_INPUT
	LRSETPOS : LREAL;
	LRSETVEL : LREAL;
	LRSETACC : LREAL;
END_VAR
VAR_IN_OUT
	AXIS : Axis_Ref;
END_VAR
END_METHOD

METHOD GETOFFSETVALUES
VAR_OUTPUT
	LROFFSETPOS : LREAL;
	LROFFSETVEL : LREAL;
	LROFFSETACC : LREAL;
END_VAR
END_METHOD

(* ---- L_MC1P_CONFIG_94HL_ETC.pou ---- *)
FUNCTION_BLOCK L_MC1P_CONFIG_94HL_ETC EXTENDS L_MC1P_Config_Drive
VAR
	STAPPLICATIONVERSION : STRING(255);
	DWAPPLICATIONVERSION : DWORD;
	DWRATEDPOWER : DWORD;
	XSETSPEEDLIMITSTOSDODEFAULT : BOOL;
END_VAR
END_FUNCTION_BLOCK

METHOD ACYCLICACTION2
VAR_IN_OUT
	AXIS : _AXIS_REF_REAL;
END_VAR
END_METHOD

(* ---- L_MC1P_CONFIG_DRIVE.pou ---- *)
FUNCTION_BLOCK L_MC1P_CONFIG_DRIVE
VAR_INPUT
	XEXECUTE : BOOL;
END_VAR
VAR_OUTPUT
	XDONE : BOOL;
	XERROR : BOOL;
	XBUSY : BOOL;
	EERRORID : WORD;
END_VAR
VAR
	XEXECUTEOLD : BOOL;
	ISTATE : INT;
	XWAITFORPARAMETERWRITEDONE : BOOL;
	XWAITFORPARAMETERREADDONE : BOOL;
	WRITEPARAMETER : L_DCO.L_DCO_WriteDriveParameter;
	READPARAMETER : L_DCO.L_DCO_ReadDriveParameter;
	READSTRINGPARAMETER : L_DCO.L_DCO_ReadDriveParameterString;
	XTESTPARAMETEREXISTING : BOOL;
	DWREADDATA : DWORD;
	SREADDATA : STRING(255);
	XREADSTRING : BOOL;
	BYSDORETRYCOUNTER : BYTE;
	IREADCOMPONENTDATASTATE : INT;
	XREADCOMPONENTDATAACTIVE : BOOL;
	WGAINCHARIDX : WORD;
	CONFIGINFO : L_MC1P_AdditionalConfigInfo;
	WOFFSET : WORD;
	SDO_WRITE_TIME_OUT : UDINT := 10000;
	SDO_READ_TIME_OUT : UDINT := 5000;
	MAX_SDO_RETRIES : BYTE := 3;
END_VAR
END_FUNCTION_BLOCK

METHOD ACYCLICACTION2
VAR_IN_OUT
	AXIS : _AXIS_REF_REAL;
END_VAR
END_METHOD

METHOD ACYCLICACTION
END_METHOD

METHOD DOFUNCTION : BOOL
VAR_INPUT
	XEXECUTE : BOOL;
	WOFFSET : WORD;
END_VAR
VAR_OUTPUT
	XDONE : BOOL;
	XERROR : BOOL;
	XBUSY : BOOL;
	EERRORID : WORD;
END_VAR
VAR_IN_OUT
	AXIS : _AXIS_REF_REAL;
END_VAR
END_METHOD

METHOD GETADDITIONALCONFIGINFO : POINTER TO L_MC1P_AdditionalConfigInfo
END_METHOD

METHOD GETCOMPONENTINFOINDEX : WORD
VAR_INPUT
	DATASELECTION : WORD;
END_VAR
VAR_OUTPUT
	USISUB : USINT;
	XISSTRING : BOOL;
END_VAR
END_METHOD

METHOD GETINSTANCE : POINTER TO BYTE
END_METHOD

METHOD READCMPINFO : BOOL
VAR_IN_OUT
	AXIS : _AXIS_REF_REAL;
END_VAR
END_METHOD

METHOD RESET : BOOL
END_METHOD

METHOD FB_INIT : BOOL
VAR_INPUT
	BINITRETAINS : BOOL;
	BINCOPYCODE : BOOL;
END_VAR
END_METHOD

(* ---- L_MC1P_CONFIG_GENERICDRIVE.pou ---- *)
FUNCTION_BLOCK L_MC1P_CONFIG_GENERICDRIVE EXTENDS L_MC1P_Config_Drive
VAR_INPUT
	ITFGENERICCONFIG : L_MC1P_IGenericAxisConfiguration;
END_VAR
VAR
	LRTORQUETEMP : LREAL;
	PGENERICAXISCONFIGURATION : POINTER TO L_MC1P_GenericAxisConfiguration;
	WEXTERNALSTEP : WORD;
END_VAR
END_FUNCTION_BLOCK

METHOD ACYCLICACTION2
VAR_IN_OUT
	AXIS : _AXIS_REF_REAL;
END_VAR
END_METHOD

(* ---- L_MC1P_CONFIG_I500.pou ---- *)
FUNCTION_BLOCK L_MC1P_CONFIG_I500 EXTENDS L_MC1P_Config_Drive
END_FUNCTION_BLOCK

METHOD ACYCLICACTION2
VAR_IN_OUT
	AXIS : _AXIS_REF_REAL;
END_VAR
END_METHOD

METHOD GETCOMPONENTINFOINDEX : WORD
VAR_INPUT
	DATASELECTION : WORD;
END_VAR
VAR_OUTPUT
	USISUB : USINT;
	XISSTRING : BOOL;
END_VAR
END_METHOD

(* ---- L_MC1P_CONFIG_I700_ETC.pou ---- *)
FUNCTION_BLOCK L_MC1P_CONFIG_I700_ETC EXTENDS L_MC1P_Config_Drive
VAR
	LRWAITCOUNTER : LREAL;
END_VAR
END_FUNCTION_BLOCK

METHOD ACYCLICACTION2
VAR_IN_OUT
	AXIS : _AXIS_REF_REAL;
END_VAR
END_METHOD

(* ---- L_MC1P_CONFIG_I900_DRIVE.pou ---- *)
FUNCTION_BLOCK L_MC1P_CONFIG_I900_DRIVE EXTENDS L_MC1P_Config_Drive
VAR_INPUT
	XINITFORCIA402AXIS : BOOL := FALSE;
END_VAR
VAR
	LRWAITCOUNTER : LREAL;
END_VAR
END_FUNCTION_BLOCK

METHOD ACYCLICACTION2
VAR_IN_OUT
	AXIS : _AXIS_REF_REAL;
END_VAR
END_METHOD

(* ---- L_MC1P_CONFIG_I900_ENC_DRIVE.pou ---- *)
FUNCTION_BLOCK L_MC1P_CONFIG_I900_ENC_DRIVE EXTENDS L_MC1P_Config_Drive
VAR
	DWENCODERSELECTION : DWORD;
	LRWAITCOUNTER : LREAL;
END_VAR
END_FUNCTION_BLOCK

METHOD ACYCLICACTION2
VAR_IN_OUT
	AXIS : _AXIS_REF_REAL;
END_VAR
END_METHOD

(* ---- L_MC1P_CONFIG_I900ADV_ETC.pou ---- *)
FUNCTION_BLOCK L_MC1P_CONFIG_I900ADV_ETC EXTENDS L_MC1P_Config_Drive
VAR_INPUT
	XCIA402ADVANCED : BOOL;
END_VAR
VAR
	DILOADFEEDCONST : DINT;
	DWLOADGEARNUM : DWORD;
	DWLOADGEARDEN : DWORD;
	LRWAITCOUNTER : LREAL;
END_VAR
END_FUNCTION_BLOCK

METHOD ACYCLICACTION2
VAR_IN_OUT
	AXIS : _AXIS_REF_REAL;
END_VAR
END_METHOD

(* ---- L_MC1P_CONSIDERMASTERUNSTEADY.pou ---- *)
FUNCTION_BLOCK L_MC1P_CONSIDERMASTERUNSTEADY
VAR_OUTPUT
	XSETVALUEMODE2POS : BOOL;
	XRECEIVEDHOMINGGAP : BOOL;
	LROFFSETATHOMINGGAP : LREAL;
	XRECEIVEDREALGAP : BOOL;
	LROFFSETATREALGAP : LREAL;
END_VAR
VAR
	_XLASTSTEADYSTATEVALID : BOOL := FALSE;
	_LRMASTERPOSITIONEXTRAPOLATE : LREAL;
	_PSTEADYSTATE : POINTER TO L_MC1P_SteadyState;
	_DWCURRENTSTEADYSTATE : DWORD;
	XLASTSTEADYSTATEVALID : BOOL;
	DWLASTSTEADYSTATE : DWORD;
	LRPOSITIONEXTRAPOLATE : LREAL;
	LRPOSITION_LAST : LREAL;
	LRTASKCYCLE : LREAL := 0;
	XREADYFORCORRREALGAP : BOOL;
	AXRECEIVEDREALGAP_LAST : ARRAY [1..2] OF BOOL;
	LRYFACTOR : LREAL;
	LRXFACTOR : LREAL;
	LRXSCALED : LREAL;
	LRYSCALED : LREAL;
	LRSETTIMECONTER : LREAL;
	LRMAXTIME : LREAL := 0.1;
	C_ALRKOEF_0_1 : ARRAY [0..5] OF LREAL := [0, 0, 0, 10, -15, 6];
END_VAR
END_FUNCTION_BLOCK

METHOD CALCFOLLOWPOSITIONGAP : BOOL
VAR_INPUT
	ESLAVETRAVERSINGRANGE : L_MC1P_TraversingRange;
	LRSLAVECYCLELENGTH : LREAL;
	LRSLAVESETVEL : LREAL;
	LRPOSITION : LREAL;
	ESETVALUEMODE : L_MC1P_SetValueMode;
END_VAR
END_METHOD

METHOD CONSIDERUNSTEADYEVENT : BOOL
VAR_INPUT
	XAXISVALID : BOOL;
	ITFMASTERVALUES : L_MC1P_IAXIS_REF_MASTERVALUES;
	ESETVALUEMODE : L_MC1P_SetValueMode;
END_VAR
END_METHOD

METHOD CORRREALGAP
END_METHOD

METHOD INITHOMINGGAP : BOOL
END_METHOD

METHOD INITREALGAP : BOOL
END_METHOD

METHOD INITIALIZE : BOOL
END_METHOD

METHOD RESETRECEIVEDGAPSTATE : BOOL
END_METHOD

(* ---- L_MC1P_CONTROLSETVALUES.pou ---- *)
FUNCTION_BLOCK L_MC1P_CONTROLSETVALUES EXTENDS L_MC1P_Template_Licence_150
VAR_INPUT
	XENABLE : BOOL;
	LRPOSITION : LREAL;
	LRVELOCITY : LREAL;
	LRACCELERATION : LREAL;
	ESETVALUEMODE : L_MC1P_SetValueMode := L_MC1P_SetValueMode.Pos;
	XIGNOREACCFORPOSCALC : BOOL;
END_VAR
VAR_OUTPUT
	XBUSY : BOOL;
	XCOMMANDABORTED : BOOL;
	XERROR : BOOL;
	EERRORID : L_IE1P_Error;
END_VAR
VAR
	FSV : L_MC1P_FollowSetValues_internal;
	XENABLEOLD : BOOL;
	WFUNID : WORD;
	XMASTERVALID : BOOL;
	XSLAVEVALID : BOOL;
	FBCONSIDERUNSTADYSLAVE : L_MC1P_ConsiderMasterUnsteady;
	FBCONSIDERUNSTADYMASTER : L_MC1P_ConsiderMasterUnsteady;
	MASTER : L_MC1P_IAXIS_REF_MASTERVALUES;
END_VAR
END_FUNCTION_BLOCK

(* ---- L_MC1P_CRITICALSECTION.pou ---- *)
FUNCTION_BLOCK L_MC1P_CRITICALSECTION EXTENDS L_UBUP_Criticalsection
END_FUNCTION_BLOCK

METHOD LOCK : BOOL
END_METHOD

METHOD LOCKSTATE : BOOL
END_METHOD

METHOD UNLOCK : BOOL
END_METHOD

(* ---- L_MC1P_CYCLICPARAMETERACCESSREAD.pou ---- *)
FUNCTION_BLOCK L_MC1P_CYCLICPARAMETERACCESSREAD EXTENDS L_MC1P_Template
VAR_INPUT
	XENABLE : BOOL;
	WINDEX : WORD;
	USISUBINDEX : USINT;
	USISIZE : USINT;
	XSIGNED : BOOL := FALSE;
	LRSCALEFACTOR : LREAL := 1;
END_VAR
VAR_OUTPUT
	XVALID : BOOL;
	XBUSY : BOOL;
	XERROR : BOOL;
	EERRORID : L_IE1P_Error;
	LRDATA : LREAL;
END_VAR
VAR
	XENABLEOLD : BOOL;
	XWAITINITVARACCESS : BOOL;
	PDATA : POINTER TO BYTE;
	PADDDATA : POINTER TO BYTE;
	PSIDUMMY : POINTER TO SINT;
	PIDUMMY : POINTER TO INT;
	PDIDUMMY : POINTER TO DINT;
	PLIDUMMY : POINTER TO LINT;
	PUSIDUMMY : POINTER TO USINT;
	PUIDUMMY : POINTER TO UINT;
	PUDIDUMMY : POINTER TO UDINT;
	PULIDUMMY : POINTER TO ULINT;
	PAXIS : POINTER TO _AXIS_REF_REAL;
	WINDEXOLD : WORD;
	USISUBINDEXOLD : USINT;
	XSUPPORTBYAXIS : BOOL;
	USISIZEINT : USINT;
	XRETRIGGERREQUEST : BOOL;
	XSENDERRORWHENAXISAVAILABLE : BOOL;
END_VAR
END_FUNCTION_BLOCK

(* ---- L_MC1P_CYCLICPARAMETERACCESSWRITE.pou ---- *)
FUNCTION_BLOCK L_MC1P_CYCLICPARAMETERACCESSWRITE EXTENDS L_MC1P_Template
VAR_INPUT
	XENABLE : BOOL;
	WINDEX : WORD;
	USISUBINDEX : USINT;
	USISIZE : USINT;
	XSIGNED : BOOL := FALSE;
	LRSCALEFACTOR : LREAL := 1;
	LRDATA : LREAL;
END_VAR
VAR_OUTPUT
	XVALID : BOOL;
	XBUSY : BOOL;
	XERROR : BOOL;
	EERRORID : L_IE1P_Error;
END_VAR
VAR
	XENABLEOLD : BOOL;
	XWAITINITVARACCESS : BOOL;
	PDATA : POINTER TO BYTE;
	PADDDATA : POINTER TO BYTE;
	PSIDUMMY : POINTER TO SINT;
	PIDUMMY : POINTER TO INT;
	PDIDUMMY : POINTER TO DINT;
	PUSIDUMMY : POINTER TO USINT;
	PUIDUMMY : POINTER TO UINT;
	PUDIDUMMY : POINTER TO UDINT;
	LRTEMP : LREAL;
	WINDEXOLD : WORD;
	USISUBINDEXOLD : USINT;
	XSUPPORTBYAXIS : BOOL;
	USISIZEINT : USINT;
	XRETRIGGERREQUEST : BOOL;
END_VAR
END_FUNCTION_BLOCK

(* ---- L_MC1P_DATAMANAGER.pou ---- *)
FUNCTION_BLOCK L_MC1P_DATAMANAGER
VAR
	PAPPLICATION : POINTER TO APPLICATION;
END_VAR
END_FUNCTION_BLOCK

METHOD AFTERWRITEOUTPUTS : INT
END_METHOD

METHOD INITIALIZE : UDINT
VAR_INPUT
	WMODULETYPE : UINT;
	DWINSTANCE : UDINT;
	PCONNECTOR : POINTER TO IoConfigConnector;
END_VAR
END_METHOD

(* ---- L_MC1P_DELAYCOMP.pou ---- *)
FUNCTION_BLOCK L_MC1P_DELAYCOMP
VAR_INPUT
	LRCYCPOSIN : LREAL;
	LRCOMPTIME : LREAL;
	LRCYCLELENGTH : LREAL;
END_VAR
VAR_OUTPUT
	LRSETPOSOUT : LREAL;
END_VAR
VAR
	LRPOS : LREAL;
	LROLDPOS : LREAL;
	LRDIFF : LREAL;
	LRFACTOR : LREAL;
	LRTASKCYCLE : LREAL;
END_VAR
END_FUNCTION_BLOCK

(* ---- L_MC1P_DELAYSETVALUES.pou ---- *)
FUNCTION_BLOCK L_MC1P_DELAYSETVALUES EXTENDS L_MC1P_SetSetValueManipulator
VAR_INPUT
	LRDELAYTIME : LREAL := 0.1;
END_VAR
VAR_OUTPUT
	XINEQOUT : BOOL;
END_VAR
VAR
	LRDELAYTIMEINT : LREAL;
	DIBUFFERINDEX : DINT;
	DIVALIDCOUNTER : DINT;
	ALRPOS : ARRAY [1..wBufferSize] OF LREAL;
	DIDELAY : DINT;
	LRPOSOUTSAVE : LREAL;
	LRPOSOUTOLD : LREAL;
	LRVELOUTOLD : LREAL;
	WBUFFERSIZE : WORD := 1000;
END_VAR
END_FUNCTION_BLOCK

METHOD RESETOUTPUTS
END_METHOD

METHOD CALCFILTERVALUES
VAR_IN_OUT
	AXIS : Axis_REf;
END_VAR
END_METHOD

METHOD READINPUTDATA
VAR_IN_OUT
	AXIS : Axis_REf;
END_VAR
END_METHOD

METHOD CALCULATE2
VAR_IN_OUT
	AXIS : Axis_REf;
END_VAR
END_METHOD

METHOD ENABLEINIT2
VAR_IN_OUT
	AXIS : Axis_REf;
END_VAR
END_METHOD

METHOD LOADOFFSET2
VAR_INPUT
	OFFSET : LREAL;
END_VAR
VAR_IN_OUT
	AXIS : Axis_REf;
END_VAR
END_METHOD

(* ---- L_MC1P_DELAYSETVALUES2.pou ---- *)
FUNCTION_BLOCK L_MC1P_DELAYSETVALUES2 EXTENDS L_MC1P_SetSetValueManipulator
VAR_INPUT
	LRDELAYTIME : LREAL := 0.1;
	XEXECUTIONINDEXINTERN : BOOL;
END_VAR
VAR
	LRDELAYTIMEINT : LREAL;
	WBUFFERINDEX : WORD;
	DIVALIDCOUNTER : DINT;
	DIDELAYPOST : DINT;
	DIDELAYPRE : DINT;
	LRDELAYPOST : LREAL;
	LRPOSOUTSAVE : LREAL;
	LRVELOUTSAVE : LREAL;
	LRACCOUTSAVE : LREAL;
	LRTORQUEOUTSAVE : LREAL;
	LRTIMEFKT : LREAL;
	SYNCTIME : DINT;
	LRPOSOUT_OLD : LREAL;
	LRVELOUT_OLD : LREAL;
	LRACCOUT_OLD : LREAL;
	LRTORQUEOUT_OLD : LREAL;
	LRTASKCYCLE : LREAL;
	LRINVTASKCYCLE : LREAL;
	WDX : WORD;
	LRCYCLELENGTH : LREAL;
	XTESTSTARTFILTER : BOOL;
	LRHOMINGOFFSETACT : LREAL;
	L_MC1P_EXTRA_INTERPOLATION1 : L_MC1P_Extra_Interpolation;
	WBUFFERSIZE : WORD := 31;
END_VAR
END_FUNCTION_BLOCK

METHOD LOADOFFSET2
VAR_INPUT
	OFFSET : LREAL;
END_VAR
VAR_IN_OUT
	AXIS : AXIS_REF;
END_VAR
END_METHOD

METHOD RESETOUTPUTS
END_METHOD

METHOD CALCULATE2
VAR_IN_OUT
	AXIS : Axis_REf;
END_VAR
END_METHOD

METHOD CONNECTTOAXIS
VAR_IN_OUT
	AXIS : Axis_Ref;
END_VAR
END_METHOD

METHOD DISCONNECTFROMAXIS
VAR_IN_OUT
	AXIS : Axis_Ref;
END_VAR
END_METHOD

METHOD ENABLEINIT2
VAR_IN_OUT
	AXIS : Axis_REf;
END_VAR
END_METHOD

METHOD READINPUTDATA
VAR_IN_OUT
	AXIS : Axis_REf;
END_VAR
END_METHOD

METHOD FILTERSTARTCONDITION
VAR_INPUT
	LRSETPOS : LREAL;
	LRSETVEL : LREAL;
	LRSETACC : LREAL;
END_VAR
VAR_IN_OUT
	AXIS : Axis_Ref;
END_VAR
END_METHOD

(* ---- L_MC1P_DISABLESWLIMIT.pou ---- *)
FUNCTION_BLOCK L_MC1P_DISABLESWLIMIT EXTENDS L_MC1P_Template
VAR_INPUT
	XENABLE : BOOL;
END_VAR
VAR_OUTPUT
	XBUSY : BOOL;
	XERROR : BOOL;
	EERRORID : L_IE1P_Error;
END_VAR
VAR
	XENABLEOLD : BOOL := FALSE;
END_VAR
END_FUNCTION_BLOCK

(* ---- L_MC1P_DRIVEERRVALUEREADER.pou ---- *)
FUNCTION_BLOCK L_MC1P_DRIVEERRVALUEREADER
VAR_INPUT
	XAXISERRORNEW : BOOL := FALSE;
	XAXISERROROLD : BOOL := FALSE;
END_VAR
VAR_OUTPUT
	DWVALUE : DWORD;
	XDONE : BOOL;
	XERROR : BOOL;
	XISPDOMAPPED : BOOL;
END_VAR
VAR
	PAXIS : POINTER TO _AXIS_REF_REAL;
	READSDO : L_DCO.L_DCO_ReadDriveParameter;
	XINITDONE : BOOL;
	BEXE : BOOL := FALSE;
	STRNAMEETCSLAVE : STRING(80);
END_VAR
END_FUNCTION_BLOCK

METHOD CYCLIC : BOOL
END_METHOD

METHOD INIT : BOOL
VAR_INPUT
	PTHEAXIS : POINTER TO _AXIS_REF_REAL;
	UIINDEX : UINT;
	USISUBINDEX : USINT;
	STRNAME : STRING(80);
END_VAR
END_METHOD

METHOD INIT_FORPDOMAPPING
VAR_INPUT
	AXIS : POINTER TO _AXIS_REF_REAL;
END_VAR
END_METHOD

METHOD INIT_FORSDOMAPPING
VAR_INPUT
	AXIS : POINTER TO _AXIS_REF_REAL;
	UIINDEX : UINT;
	USISUBINDEX : USINT;
END_VAR
END_METHOD

(* ---- L_MC1P_DRIVESCALING.pou ---- *)
FUNCTION_BLOCK L_MC1P_DRIVESCALING
END_FUNCTION_BLOCK

METHOD CALCACCFACTOR : BOOL
VAR_OUTPUT
	LRSCALEUNITTOACC : LREAL;
	LRSCALEACCTOUNIT : LREAL;
END_VAR
VAR_IN_OUT
	AXIS : _AXIS_REF_REAL;
END_VAR
END_METHOD

METHOD CALCSPEEDFACTOR : BOOL
VAR_OUTPUT
	LRSCALEUNITTOSPEED : LREAL;
	LRSCALESPEEDTOUNIT : LREAL;
END_VAR
VAR_IN_OUT
	AXIS : _AXIS_REF_REAL;
END_VAR
END_METHOD

METHOD CALCTORQUEFACTOR : BOOL
VAR_OUTPUT
	LRSCALETORQUETONORM : LREAL;
	LRSCALETORQUETONORM2 : LREAL;
	LRSCALENORMTOTORQUE : LREAL;
END_VAR
VAR_IN_OUT
	AXIS : _AXIS_REF_REAL;
END_VAR
END_METHOD

METHOD CHECKVALIDPOSRESOLUTION : BOOL
VAR_INPUT
	DWPOSRESOLUTION : DWORD;
END_VAR
END_METHOD

METHOD GETDEFAULTTORQUE : LREAL
VAR_INPUT
	LRREFTORQUE : LREAL;
END_VAR
END_METHOD

METHOD POSDIFFTOSPEEDINC : DINT
VAR_INPUT
	DIPOSDIFF : DINT := 0;
	DWFACTOR : DWORD := 1000;
END_VAR
VAR_IN_OUT
	AXIS : _AXIS_REF_REAL;
END_VAR
END_METHOD

METHOD SPEEDTOPOSDIFFINC : DINT
VAR_INPUT
	DISPEED : DINT := 0;
	DWFACTOR : DWORD := 1000;
END_VAR
VAR_IN_OUT
	AXIS : _AXIS_REF_REAL;
	DIRES : DINT;
END_VAR
END_METHOD

(* ---- L_MC1P_DRIVESCALING_94HL.pou ---- *)
FUNCTION_BLOCK L_MC1P_DRIVESCALING_94HL
END_FUNCTION_BLOCK

METHOD CALCACCFACTOR : BOOL
VAR_OUTPUT
	LRSCALEUNITTOACC : LREAL;
	LRSCALEACCTOUNIT : LREAL;
END_VAR
VAR_IN_OUT
	AXIS : _AXIS_REF_REAL;
END_VAR
END_METHOD

METHOD CALCSPEEDFACTOR : BOOL
VAR_OUTPUT
	LRSCALEUNITTOSPEED : LREAL;
	LRSCALESPEEDTOUNIT : LREAL;
END_VAR
VAR_IN_OUT
	AXIS : _AXIS_REF_REAL;
END_VAR
END_METHOD

METHOD CALCTORQUEFACTOR : BOOL
VAR_OUTPUT
	LRSCALETORQUETONORM : LREAL;
	LRSCALETORQUETONORM2 : LREAL;
	LRSCALENORMTOTORQUE : LREAL;
END_VAR
VAR_IN_OUT
	AXIS : _AXIS_REF_REAL;
END_VAR
END_METHOD

METHOD CHECKVALIDPOSRESOLUTION : BOOL
VAR_INPUT
	DWPOSRESOLUTION : DWORD;
END_VAR
END_METHOD

METHOD GETDEFAULTTORQUE : LREAL
VAR_INPUT
	LRREFTORQUE : LREAL;
END_VAR
END_METHOD

METHOD POSDIFFTOSPEEDINC : DINT
VAR_INPUT
	DIPOSDIFF : DINT := 0;
	DWFACTOR : DWORD := 1000;
END_VAR
VAR_IN_OUT
	AXIS : _AXIS_REF_REAL;
END_VAR
END_METHOD

METHOD SPEEDTOPOSDIFFINC : DINT
VAR_INPUT
	DISPEED : DINT := 0;
	DWFACTOR : DWORD := 1000;
END_VAR
VAR_IN_OUT
	AXIS : _AXIS_REF_REAL;
	DIRES : DINT;
END_VAR
END_METHOD
